LIN {X 0,Y 523.904,Z 128.222,A -85,B 0,C 180,E1 -4806.401,E2 -4806.401} C_VEL
LIN {X 0,Y 523.923,Z 128.218,A -85,B 0,C 180,E1 -4809.084,E2 -4809.084} C_VEL
LIN {X 0,Y 523.952,Z 128.218,A -85,B 0,C 180,E1 -4812.119,E2 -4812.119} C_VEL
LIN {X 0,Y 523.947,Z 128.218,A -85,B 0,C 180,E1 -4815.31,E2 -4815.31} C_VEL
LIN {X 0,Y 523.956,Z 128.214,A -85,B 0,C 180,E1 -4818.69,E2 -4818.69} C_VEL
LIN {X 0,Y 523.918,Z 128.221,A -85,B 0,C 180,E1 -4821.08,E2 -4821.08} C_VEL
LIN {X 0,Y 523.901,Z 128.225,A -85,B 0,C 180,E1 -4823.825,E2 -4823.825} C_VEL
LIN {X 0,Y 523.913,Z 128.219,A -85,B 0,C 180,E1 -4826.633,E2 -4826.633} C_VEL
LIN {X 0,Y 523.949,Z 128.223,A -85,B 0,C 180,E1 -4829.355,E2 -4829.355} C_VEL
LIN {X 0,Y 523.977,Z 128.211,A -85,B 0,C 180,E1 -4832.281,E2 -4832.281} C_VEL
LIN {X 0,Y 523.953,Z 128.215,A -85,B 0,C 180,E1 -4834.581,E2 -4834.581} C_VEL
LIN {X 0,Y 523.912,Z 128.227,A -85,B 0,C 180,E1 -4837.106,E2 -4837.106} C_VEL
LIN {X 0,Y 523.979,Z 128.211,A -85,B 0,C 180,E1 -4839.866,E2 -4839.866} C_VEL
LIN {X 0,Y 523.956,Z 128.219,A -85,B 0,C 180,E1 -4842.837,E2 -4842.837} C_VEL
LIN {X 0,Y 523.978,Z 128.217,A -85,B 0,C 180,E1 -4845.236,E2 -4845.236} C_VEL
LIN {X 0,Y 524.013,Z 128.208,A -85,B 0,C 180,E1 -4848.394,E2 -4848.394} C_VEL
LIN {X 0,Y 523.988,Z 128.211,A -85,B 0,C 180,E1 -4851.516,E2 -4851.516} C_VEL
LIN {X 0,Y 524.08,Z 128.204,A -85,B 0,C 180,E1 -4854.613,E2 -4854.613} C_VEL
LIN {X 0,Y 524.112,Z 128.194,A -85,B 0,C 180,E1 -4857.694,E2 -4857.694} C_VEL
LIN {X 0,Y 524.123,Z 128.2,A -85,B 0,C 180,E1 -4860.768,E2 -4860.768} C_VEL
LIN {X 0,Y 524.069,Z 128.202,A -85,B 0,C 180,E1 -4863.075,E2 -4863.075} C_VEL
LIN {X 0,Y 524.037,Z 128.207,A -85,B 0,C 180,E1 -4866.159,E2 -4866.159} C_VEL
LIN {X 0,Y 524,Z 128.217,A -85,B 0,C 180,E1 -4868.484,E2 -4868.484} C_VEL
LIN {X 0,Y 524.003,Z 128.209,A -85,B 0,C 180,E1 -4871.739,E2 -4871.739} C_VEL
LIN {X 0,Y 523.993,Z 128.21,A -85,B 0,C 180,E1 -4875.052,E2 -4875.052} C_VEL
LIN {X 0,Y 523.947,Z 128.219,A -85,B 0,C 180,E1 -4877.969,E2 -4877.969} C_VEL
LIN {X 0,Y 523.971,Z 128.218,A -85,B 0,C 180,E1 -4880.41,E2 -4880.41} C_VEL
LIN {X 0,Y 523.91,Z 128.22,A -85,B 0,C 180,E1 -4882.893,E2 -4882.893} C_VEL
LIN {X 0,Y 523.983,Z 128.218,A -85,B 0,C 180,E1 -4886.02,E2 -4886.02} C_VEL
LIN {X 0,Y 523.928,Z 128.217,A -85,B 0,C 180,E1 -4888.875,E2 -4888.875} C_VEL
LIN {X 0,Y 523.92,Z 128.221,A -85,B 0,C 180,E1 -4891.544,E2 -4891.544} C_VEL
LIN {X 0,Y 523.932,Z 128.22,A -85,B 0,C 180,E1 -4894.29,E2 -4894.29} C_VEL
LIN {X 0,Y 523.906,Z 128.221,A -85,B 0,C 180,E1 -4897.132,E2 -4897.132} C_VEL
LIN {X 0,Y 523.937,Z 128.22,A -85,B 0,C 180,E1 -4900.13,E2 -4900.13} C_VEL
LIN {X 0,Y 523.92,Z 128.22,A -85,B 0,C 180,E1 -4903.167,E2 -4903.167} C_VEL
LIN {X 0,Y 523.935,Z 128.223,A -85,B 0,C 180,E1 -4905.772,E2 -4905.772} C_VEL
LIN {X 0,Y 523.918,Z 128.219,A -85,B 0,C 180,E1 -4906.912,E2 -4906.912} C_VEL
LIN {X 0,Y 523.25,Z 128.31,A -85,B 0,C 180,E1 -4907.554,E2 -4907.554} C_VEL
LIN {X 0,Y 520.408,Z 128.661,A -85,B 0,C 180,E1 -4908.596,E2 -4908.596} C_VEL
LIN {X 0,Y 518.004,Z 128.962,A -85,B 0,C 180,E1 -4909.434,E2 -4909.434} C_VEL
LIN {X 0,Y 516.967,Z 129.086,A -85,B 0,C 180,E1 -4910.082,E2 -4910.082} C_VEL
LIN {X 0,Y 516.88,Z 129.096,A -85,B 0,C 180,E1 -4910.301,E2 -4910.301} C_VEL
LIN {X 0,Y 516.876,Z 129.103,A -85,B 0,C 180,E1 -4913.343,E2 -4913.343} C_VEL
LIN {X 0,Y 516.883,Z 129.095,A -85,B 0,C 180,E1 -4916.119,E2 -4916.119} C_VEL
LIN {X 0,Y 516.889,Z 129.097,A -85,B 0,C 180,E1 -4918.936,E2 -4918.936} C_VEL
LIN {X 0,Y 516.915,Z 129.095,A -85,B 0,C 180,E1 -4921.585,E2 -4921.585} C_VEL
LIN {X 0,Y 516.931,Z 129.089,A -85,B 0,C 180,E1 -4924.211,E2 -4924.211} C_VEL
LIN {X 0,Y 516.864,Z 129.101,A -85,B 0,C 180,E1 -4926.776,E2 -4926.776} C_VEL
LIN {X 0,Y 516.939,Z 129.089,A -85,B 0,C 180,E1 -4929.732,E2 -4929.732} C_VEL
LIN {X 0,Y 516.906,Z 129.095,A -85,B 0,C 180,E1 -4932.596,E2 -4932.596} C_VEL
LIN {X 0,Y 516.941,Z 129.096,A -85,B 0,C 180,E1 -4935.03,E2 -4935.03} C_VEL
LIN {X 0,Y 516.966,Z 129.085,A -85,B 0,C 180,E1 -4938.234,E2 -4938.234} C_VEL
LIN {X 0,Y 516.956,Z 129.087,A -85,B 0,C 180,E1 -4941.4,E2 -4941.4} C_VEL
LIN {X 0,Y 517.027,Z 129.082,A -85,B 0,C 180,E1 -4944.54,E2 -4944.54} C_VEL
LIN {X 0,Y 517.084,Z 129.072,A -85,B 0,C 180,E1 -4947.663,E2 -4947.663} C_VEL
LIN {X 0,Y 517.089,Z 129.079,A -85,B 0,C 180,E1 -4950.779,E2 -4950.779} C_VEL
LIN {X 0,Y 517.058,Z 129.277,A -85,B 0,C 180,E1 -4950.925,E2 -4950.925} C_VEL
LIN {X 0,Y 517.506,Z 134.385,A -85,B 0,C 180,E1 -4951.946,E2 -4951.946} C_VEL
LIN {X 0,Y 517.261,Z 148.661,A -85,B 0,C 180,E1 -4954.701,E2 -4954.701} C_VEL
LIN {X 0,Y 519.14,Z 158.814,A -85,B 0,C 180,E1 -4954.902,E2 -4954.902} C_VEL
LIN {X 0,Y 518.601,Z 255.581,A -85,B 0,C 180,E1 -4956.273,E2 -4956.273} C_VEL
LIN {X 0,Y 518.422,Z 269.344,A -85,B 0,C 180,E1 -4956.642,E2 -4956.642} C_VEL
LIN {X 0,Y 518.231,Z 280.872,A -85,B 0,C 180,E1 -4957.097,E2 -4957.097} C_VEL
LIN {X 0,Y 518.001,Z 292.37,A -85,B 0,C 180,E1 -4957.702,E2 -4957.702} C_VEL
LIN {X 0,Y 517.716,Z 303.803,A -85,B 0,C 180,E1 -4958.48,E2 -4958.48} C_VEL
LIN {X 0,Y 517.374,Z 314.408,A -85,B 0,C 180,E1 -4959.382,E2 -4959.382} C_VEL
LIN {X 0,Y 517.083,Z 323.83,A -85,B 0,C 180,E1 -4960.375,E2 -4960.375} C_VEL
LIN {X 0,Y 516.843,Z 333.07,A -85,B 0,C 180,E1 -4961.592,E2 -4961.592} C_VEL
LIN {X 0,Y 516.622,Z 340.269,A -85,B 0,C 180,E1 -4962.772,E2 -4962.772} C_VEL
LIN {X 0,Y 516.533,Z 345.22,A -85,B 0,C 180,E1 -4963.775,E2 -4963.775} C_VEL
LIN {X 0,Y 516.432,Z 350.035,A -85,B 0,C 180,E1 -4964.985,E2 -4964.985} C_VEL
LIN {X 0,Y 516.314,Z 353.712,A -85,B 0,C 180,E1 -4966.203,E2 -4966.203} C_VEL
LIN {X 0,Y 516.245,Z 356.678,A -85,B 0,C 180,E1 -4967.644,E2 -4967.644} C_VEL
LIN {X 0,Y 516.206,Z 358.228,A -85,B 0,C 180,E1 -4969.072,E2 -4969.072} C_VEL
LIN {X 0,Y 516.228,Z 358.561,A -85,B 0,C 180,E1 -4970.053,E2 -4970.053} C_VEL
LIN {X 0,Y 516.211,Z 357.794,A -85,B 0,C 180,E1 -4971.567,E2 -4971.567} C_VEL
LIN {X 0,Y 516.252,Z 356.747,A -85,B 0,C 180,E1 -4972.407,E2 -4972.407} C_VEL
LIN {X 0,Y 516.322,Z 354.262,A -85,B 0,C 180,E1 -4973.675,E2 -4973.675} C_VEL
LIN {X 0,Y 516.407,Z 350.603,A -85,B 0,C 180,E1 -4974.954,E2 -4974.954} C_VEL
LIN {X 0,Y 516.519,Z 345.117,A -85,B 0,C 180,E1 -4976.348,E2 -4976.348} C_VEL
LIN {X 0,Y 516.664,Z 339.024,A -85,B 0,C 180,E1 -4977.548,E2 -4977.548} C_VEL
LIN {X 0,Y 516.848,Z 332.152,A -85,B 0,C 180,E1 -4978.641,E2 -4978.641} C_VEL
LIN {X 0,Y 517.083,Z 324.555,A -85,B 0,C 180,E1 -4979.635,E2 -4979.635} C_VEL
LIN {X 0,Y 517.367,Z 315.378,A -85,B 0,C 180,E1 -4980.624,E2 -4980.624} C_VEL
LIN {X 0,Y 517.6,Z 304.961,A -85,B 0,C 180,E1 -4981.531,E2 -4981.531} C_VEL
LIN {X 0,Y 517.962,Z 293.968,A -85,B 0,C 180,E1 -4982.294,E2 -4982.294} C_VEL
LIN {X 0,Y 518.27,Z 281.601,A -85,B 0,C 180,E1 -4982.964,E2 -4982.964} C_VEL
LIN {X 0,Y 518.469,Z 268.694,A -85,B 0,C 180,E1 -4983.472,E2 -4983.472} C_VEL
LIN {X 0,Y 518.68,Z 255.806,A -85,B 0,C 180,E1 -4983.812,E2 -4983.812} C_VEL
LIN {X 0,Y 519.059,Z 157.607,A -85,B 0,C 180,E1 -4985.21,E2 -4985.21} C_VEL
LIN {X 0,Y 517.299,Z 148.488,A -85,B 0,C 180,E1 -4985.408,E2 -4985.408} C_VEL
LIN {X 0,Y 517.5,Z 133.51,A -85,B 0,C 180,E1 -4988.302,E2 -4988.302} C_VEL
LIN {X 0,Y 516.927,Z 129.098,A -85,B 0,C 180,E1 -4989.199,E2 -4989.199} C_VEL
LIN {X 0,Y 516.85,Z 129.105,A -85,B 0,C 180,E1 -4991.782,E2 -4991.782} C_VEL
LIN {X 0,Y 516.896,Z 129.102,A -85,B 0,C 180,E1 -4995.007,E2 -4995.007} C_VEL
LIN {X 0,Y 516.855,Z 129.102,A -85,B 0,C 180,E1 -4998.406,E2 -4998.406} C_VEL
LIN {X 0,Y 516.876,Z 129.103,A -85,B 0,C 180,E1 -5001.284,E2 -5001.284} C_VEL
LIN {X 0,Y 516.865,Z 129.096,A -85,B 0,C 180,E1 -5004.219,E2 -5004.219} C_VEL
LIN {X 0,Y 516.879,Z 129.104,A -85,B 0,C 180,E1 -5007.052,E2 -5007.052} C_VEL
LIN {X 0,Y 516.843,Z 129.102,A -85,B 0,C 180,E1 -5009.793,E2 -5009.793} C_VEL
LIN {X 0,Y 516.868,Z 129.103,A -85,B 0,C 180,E1 -5012.464,E2 -5012.464} C_VEL
LIN {X 0,Y 516.842,Z 129.105,A -85,B 0,C 180,E1 -5015.068,E2 -5015.068} C_VEL
LIN {X 0,Y 516.87,Z 129.095,A -85,B 0,C 180,E1 -5017.622,E2 -5017.622} C_VEL
LIN {X 0,Y 516.862,Z 129.102,A -85,B 0,C 180,E1 -5020.127,E2 -5020.127} C_VEL
LIN {X 0,Y 516.869,Z 129.104,A -85,B 0,C 180,E1 -5022.594,E2 -5022.594} C_VEL
LIN {X 0,Y 516.873,Z 129.096,A -85,B 0,C 180,E1 -5025.028,E2 -5025.028} C_VEL
LIN {X 0,Y 516.921,Z 129.096,A -85,B 0,C 180,E1 -5028.233,E2 -5028.233} C_VEL
LIN {X 0,Y 516.917,Z 129.092,A -85,B 0,C 180,E1 -5031.399,E2 -5031.399} C_VEL
LIN {X 0,Y 516.978,Z 129.085,A -85,B 0,C 180,E1 -5034.54,E2 -5034.54} C_VEL
LIN {X 0,Y 517.073,Z 129.075,A -85,B 0,C 180,E1 -5037.663,E2 -5037.663} C_VEL
LIN {X 0,Y 517.066,Z 129.079,A -85,B 0,C 180,E1 -5040,E2 -5040} C_VEL
LIN {X 0,Y 517.073,Z 129.07,A -85,B 0,C 180,E1 -5042.337,E2 -5042.337} C_VEL
LIN {X 0,Y 516.969,Z 129.085,A -85,B 0,C 180,E1 -5046.244,E2 -5046.244} C_VEL
LIN {X 0,Y 516.913,Z 129.095,A -85,B 0,C 180,E1 -5049.39,E2 -5049.39} C_VEL
LIN {X 0,Y 516.955,Z 129.088,A -85,B 0,C 180,E1 -5051.807,E2 -5051.807} C_VEL
LIN {X 0,Y 516.939,Z 129.093,A -85,B 0,C 180,E1 -5055.143,E2 -5055.143} C_VEL
LIN {X 0,Y 516.88,Z 129.093,A -85,B 0,C 180,E1 -5058.224,E2 -5058.224} C_VEL
LIN {X 0,Y 516.907,Z 129.094,A -85,B 0,C 180,E1 -5060.702,E2 -5060.702} C_VEL
LIN {X 0,Y 516.887,Z 129.095,A -85,B 0,C 180,E1 -5064.073,E2 -5064.073} C_VEL
LIN {X 0,Y 516.896,Z 129.095,A -85,B 0,C 180,E1 -5066.66,E2 -5066.66} C_VEL
LIN {X 0,Y 516.888,Z 129.095,A -85,B 0,C 180,E1 -5069.519,E2 -5069.519} C_VEL
LIN {X 0,Y 516.896,Z 129.098,A -85,B 0,C 180,E1 -5072.543,E2 -5072.543} C_VEL
LIN {X 0,Y 516.867,Z 129.1,A -85,B 0,C 180,E1 -5075.329,E2 -5075.329} C_VEL
LIN {X 0,Y 516.881,Z 129.095,A -85,B 0,C 180,E1 -5077.943,E2 -5077.943} C_VEL
LIN {X 0,Y 516.866,Z 129.105,A -85,B 0,C 180,E1 -5080.744,E2 -5080.744} C_VEL
LIN {X 0,Y 516.857,Z 129.104,A -85,B 0,C 180,E1 -5082.834,E2 -5082.834} C_VEL
LIN {X 0,Y 516.898,Z 129.096,A -85,B 0,C 180,E1 -5085.007,E2 -5085.007} C_VEL
LIN {X 0,Y 516.911,Z 129.101,A -85,B 0,C 180,E1 -5088.4,E2 -5088.4} C_VEL
LIN {X 0,Y 516.883,Z 129.096,A -85,B 0,C 180,E1 -5091.284,E2 -5091.284} C_VEL
LIN {X 0,Y 516.87,Z 129.105,A -85,B 0,C 180,E1 -5094.219,E2 -5094.219} C_VEL
LIN {X 0,Y 516.898,Z 129.095,A -85,B 0,C 180,E1 -5097.053,E2 -5097.053} C_VEL
LIN {X 0,Y 516.889,Z 129.101,A -85,B 0,C 180,E1 -5099.796,E2 -5099.796} C_VEL
LIN {X 0,Y 516.925,Z 129.095,A -85,B 0,C 180,E1 -5102.467,E2 -5102.467} C_VEL
LIN {X 0,Y 516.941,Z 129.15,A -85,B 0,C 180,E1 -5104.939,E2 -5104.939} C_VEL
LIN {X 0,Y 518.489,Z 138.225,A -85,B 0,C 180,E1 -5106.43,E2 -5106.43} C_VEL
LIN {X 0,Y 517.938,Z 158.539,A -85,B 0,C 180,E1 -5109.543,E2 -5109.543} C_VEL
LIN {X 0,Y 517.506,Z 178.873,A -85,B 0,C 180,E1 -5112.616,E2 -5112.616} C_VEL
LIN {X 0,Y 517.216,Z 192.296,A -85,B 0,C 180,E1 -5114.623,E2 -5114.623} C_VEL
LIN {X 0,Y 519.028,Z 206.259,A -85,B 0,C 180,E1 -5114.878,E2 -5114.878} C_VEL
LIN {X 0,Y 518.589,Z 300.529,A -85,B 0,C 180,E1 -5116.206,E2 -5116.206} C_VEL
LIN {X 0,Y 518.322,Z 313.972,A -85,B 0,C 180,E1 -5116.548,E2 -5116.548} C_VEL
LIN {X 0,Y 518.034,Z 327.363,A -85,B 0,C 180,E1 -5117.065,E2 -5117.065} C_VEL
LIN {X 0,Y 517.778,Z 338.798,A -85,B 0,C 180,E1 -5117.668,E2 -5117.668} C_VEL
LIN {X 0,Y 517.447,Z 350.26,A -85,B 0,C 180,E1 -5118.443,E2 -5118.443} C_VEL
LIN {X 0,Y 517.191,Z 360.762,A -85,B 0,C 180,E1 -5119.33,E2 -5119.33} C_VEL
LIN {X 0,Y 516.899,Z 369.348,A -85,B 0,C 180,E1 -5120.215,E2 -5120.215} C_VEL
LIN {X 0,Y 516.68,Z 377.273,A -85,B 0,C 180,E1 -5121.198,E2 -5121.198} C_VEL
LIN {X 0,Y 516.516,Z 385.017,A -85,B 0,C 180,E1 -5122.376,E2 -5122.376} C_VEL
LIN {X 0,Y 516.374,Z 392.154,A -85,B 0,C 180,E1 -5123.749,E2 -5123.749} C_VEL
LIN {X 0,Y 516.312,Z 396.906,A -85,B 0,C 180,E1 -5124.924,E2 -5124.924} C_VEL
LIN {X 0,Y 516.352,Z 400.54,A -85,B 0,C 180,E1 -5126.098,E2 -5126.098} C_VEL
LIN {X 0,Y 516.303,Z 402.413,A -85,B 0,C 180,E1 -5126.879,E2 -5126.879} C_VEL
LIN {X 0,Y 516.264,Z 403.816,A -85,B 0,C 180,E1 -5127.659,E2 -5127.659} C_VEL
LIN {X 0,Y 516.172,Z 405.43,A -85,B 0,C 180,E1 -5129.22,E2 -5129.22} C_VEL
LIN {X 0,Y 516.173,Z 405.651,A -85,B 0,C 180,E1 -5130,E2 -5130} C_VEL
LIN {X 0,Y 516.193,Z 404.829,A -85,B 0,C 180,E1 -5131.56,E2 -5131.56} C_VEL
LIN {X 0,Y 516.264,Z 403.835,A -85,B 0,C 180,E1 -5132.34,E2 -5132.34} C_VEL
LIN {X 0,Y 516.303,Z 402.436,A -85,B 0,C 180,E1 -5133.121,E2 -5133.121} C_VEL
LIN {X 0,Y 516.31,Z 399.49,A -85,B 0,C 180,E1 -5134.293,E2 -5134.293} C_VEL
LIN {X 0,Y 516.367,Z 395.502,A -85,B 0,C 180,E1 -5135.467,E2 -5135.467} C_VEL
LIN {X 0,Y 516.427,Z 389.355,A -85,B 0,C 180,E1 -5136.84,E2 -5136.84} C_VEL
LIN {X 0,Y 516.567,Z 382.66,A -85,B 0,C 180,E1 -5138.016,E2 -5138.016} C_VEL
LIN {X 0,Y 516.755,Z 374.344,A -85,B 0,C 180,E1 -5139.195,E2 -5139.195} C_VEL
LIN {X 0,Y 516.985,Z 365.818,A -85,B 0,C 180,E1 -5140.179,E2 -5140.179} C_VEL
LIN {X 0,Y 517.301,Z 355.287,A -85,B 0,C 180,E1 -5141.163,E2 -5141.163} C_VEL
LIN {X 0,Y 517.621,Z 343.415,A -85,B 0,C 180,E1 -5142.051,E2 -5142.051} C_VEL
LIN {X 0,Y 517.947,Z 331.506,A -85,B 0,C 180,E1 -5142.738,E2 -5142.738} C_VEL
LIN {X 0,Y 518.211,Z 319.097,A -85,B 0,C 180,E1 -5143.28,E2 -5143.28} C_VEL
LIN {X 0,Y 518.484,Z 306.333,A -85,B 0,C 180,E1 -5143.672,E2 -5143.672} C_VEL
LIN {X 0,Y 518.634,Z 291.09,A -85,B 0,C 180,E1 -5143.943,E2 -5143.943} C_VEL
LIN {X 0,Y 518.97,Z 204.341,A -85,B 0,C 180,E1 -5145.152,E2 -5145.152} C_VEL
LIN {X 0,Y 517.23,Z 192.384,A -85,B 0,C 180,E1 -5145.39,E2 -5145.39} C_VEL
LIN {X 0,Y 517.621,Z 174.235,A -85,B 0,C 180,E1 -5148.116,E2 -5148.116} C_VEL
LIN {X 0,Y 518.165,Z 152.086,A -85,B 0,C 180,E1 -5151.482,E2 -5151.482} C_VEL
LIN {X 0,Y 518.451,Z 137.182,A -85,B 0,C 180,E1 -5153.783,E2 -5153.783} C_VEL
LIN {X 0,Y 516.924,Z 129.096,A -85,B 0,C 180,E1 -5155.142,E2 -5155.142} C_VEL
LIN {X 0,Y 516.918,Z 129.099,A -85,B 0,C 180,E1 -5157.903,E2 -5157.903} C_VEL
LIN {X 0,Y 516.894,Z 129.102,A -85,B 0,C 180,E1 -5160.203,E2 -5160.203} C_VEL
LIN {X 0,Y 516.896,Z 129.093,A -85,B 0,C 180,E1 -5162.947,E2 -5162.947} C_VEL
LIN {X 0,Y 516.872,Z 129.103,A -85,B 0,C 180,E1 -5165.78,E2 -5165.78} C_VEL
LIN {X 0,Y 516.883,Z 129.095,A -85,B 0,C 180,E1 -5168.716,E2 -5168.716} C_VEL
LIN {X 0,Y 516.913,Z 129.1,A -85,B 0,C 180,E1 -5171.775,E2 -5171.775} C_VEL
LIN {X 0,Y 516.896,Z 129.094,A -85,B 0,C 180,E1 -5175.007,E2 -5175.007} C_VEL
LIN {X 0,Y 516.914,Z 129.091,A -85,B 0,C 180,E1 -5178.399,E2 -5178.399} C_VEL
LIN {X 0,Y 516.881,Z 129.1,A -85,B 0,C 180,E1 -5181.284,E2 -5181.284} C_VEL
LIN {X 0,Y 516.871,Z 129.097,A -85,B 0,C 180,E1 -5184.219,E2 -5184.219} C_VEL
LIN {X 0,Y 516.881,Z 129.098,A -85,B 0,C 180,E1 -5187.052,E2 -5187.052} C_VEL
LIN {X 0,Y 516.887,Z 129.097,A -85,B 0,C 180,E1 -5189.796,E2 -5189.796} C_VEL
LIN {X 0,Y 516.926,Z 129.09,A -85,B 0,C 180,E1 -5192.467,E2 -5192.467} C_VEL
LIN {X 0,Y 516.909,Z 129.098,A -85,B 0,C 180,E1 -5195.072,E2 -5195.072} C_VEL
LIN {X 0,Y 516.886,Z 129.095,A -85,B 0,C 180,E1 -5198.462,E2 -5198.462} C_VEL
LIN {X 0,Y 516.9,Z 129.099,A -85,B 0,C 180,E1 -5200.955,E2 -5200.955} C_VEL
LIN {X 0,Y 516.907,Z 129.096,A -85,B 0,C 180,E1 -5203.41,E2 -5203.41} C_VEL
LIN {X 0,Y 516.894,Z 129.094,A -85,B 0,C 180,E1 -5205.833,E2 -5205.833} C_VEL
LIN {X 0,Y 516.966,Z 129.085,A -85,B 0,C 180,E1 -5208.234,E2 -5208.234} C_VEL
LIN {X 0,Y 516.956,Z 129.088,A -85,B 0,C 180,E1 -5211.399,E2 -5211.399} C_VEL
LIN {X 0,Y 517.027,Z 129.082,A -85,B 0,C 180,E1 -5214.54,E2 -5214.54} C_VEL
LIN {X 0,Y 517.084,Z 129.07,A -85,B 0,C 180,E1 -5217.663,E2 -5217.663} C_VEL
LIN {X 0,Y 517.093,Z 129.076,A -85,B 0,C 180,E1 -5220.779,E2 -5220.779} C_VEL
LIN {X 0,Y 517.01,Z 129.081,A -85,B 0,C 180,E1 -5223.117,E2 -5223.117} C_VEL
LIN {X 0,Y 517.002,Z 129.084,A -85,B 0,C 180,E1 -5226.243,E2 -5226.243} C_VEL
LIN {X 0,Y 516.945,Z 129.087,A -85,B 0,C 180,E1 -5229.389,E2 -5229.389} C_VEL
LIN {X 0,Y 516.952,Z 129.088,A -85,B 0,C 180,E1 -5231.807,E2 -5231.807} C_VEL
LIN {X 0,Y 516.944,Z 129.087,A -85,B 0,C 180,E1 -5235.146,E2 -5235.146} C_VEL
LIN {X 0,Y 516.915,Z 129.099,A -85,B 0,C 180,E1 -5238.222,E2 -5238.222} C_VEL
LIN {X 0,Y 516.912,Z 129.094,A -85,B 0,C 180,E1 -5240.701,E2 -5240.701} C_VEL
LIN {X 0,Y 516.89,Z 129.102,A -85,B 0,C 180,E1 -5244.073,E2 -5244.073} C_VEL
LIN {X 0,Y 516.921,Z 129.092,A -85,B 0,C 180,E1 -5246.658,E2 -5246.658} C_VEL
LIN {X 0,Y 516.909,Z 129.094,A -85,B 0,C 180,E1 -5249.523,E2 -5249.523} C_VEL
LIN {X 0,Y 516.895,Z 129.095,A -85,B 0,C 180,E1 -5252.543,E2 -5252.543} C_VEL
LIN {X 0,Y 516.865,Z 129.099,A -85,B 0,C 180,E1 -5255.33,E2 -5255.33} C_VEL
LIN {X 0,Y 516.88,Z 129.102,A -85,B 0,C 180,E1 -5257.943,E2 -5257.943} C_VEL
LIN {X 0,Y 516.882,Z 129.095,A -85,B 0,C 180,E1 -5260.742,E2 -5260.742} C_VEL
LIN {X 0,Y 516.883,Z 129.095,A -85,B 0,C 180,E1 -5262.831,E2 -5262.831} C_VEL
LIN {X 0,Y 516.882,Z 129.098,A -85,B 0,C 180,E1 -5266.097,E2 -5266.097} C_VEL
LIN {X 0,Y 516.912,Z 129.091,A -85,B 0,C 180,E1 -5268.399,E2 -5268.399} C_VEL
LIN {X 0,Y 516.88,Z 129.096,A -85,B 0,C 180,E1 -5270.301,E2 -5270.301} C_VEL
LIN {X 0,Y 516.209,Z 129.181,A -85,B 0,C 180,E1 -5270.952,E2 -5270.952} C_VEL
LIN {X 0,Y 513.362,Z 129.541,A -85,B 0,C 180,E1 -5272.007,E2 -5272.007} C_VEL
LIN {X 0,Y 510.952,Z 129.844,A -85,B 0,C 180,E1 -5272.857,E2 -5272.857} C_VEL
LIN {X 0,Y 509.909,Z 129.972,A -85,B 0,C 180,E1 -5273.514,E2 -5273.514} C_VEL
LIN {X 0,Y 509.819,Z 129.98,A -85,B 0,C 180,E1 -5273.736,E2 -5273.736} C_VEL
LIN {X 0,Y 509.841,Z 129.972,A -85,B 0,C 180,E1 -5276.538,E2 -5276.538} C_VEL
LIN {X 0,Y 509.842,Z 129.981,A -85,B 0,C 180,E1 -5279.334,E2 -5279.334} C_VEL
LIN {X 0,Y 509.889,Z 129.966,A -85,B 0,C 180,E1 -5282.054,E2 -5282.054} C_VEL
LIN {X 0,Y 509.875,Z 129.97,A -85,B 0,C 180,E1 -5284.704,E2 -5284.704} C_VEL
LIN {X 0,Y 509.826,Z 129.978,A -85,B 0,C 180,E1 -5287.458,E2 -5287.458} C_VEL
LIN {X 0,Y 509.916,Z 129.963,A -85,B 0,C 180,E1 -5289.845,E2 -5289.845} C_VEL
LIN {X 0,Y 509.873,Z 129.975,A -85,B 0,C 180,E1 -5293.174,E2 -5293.174} C_VEL
LIN {X 0,Y 509.861,Z 129.971,A -85,B 0,C 180,E1 -5295.634,E2 -5295.634} C_VEL
LIN {X 0,Y 509.913,Z 129.972,A -85,B 0,C 180,E1 -5298.875,E2 -5298.875} C_VEL
LIN {X 0,Y 509.921,Z 129.963,A -85,B 0,C 180,E1 -5302.078,E2 -5302.078} C_VEL
LIN {X 0,Y 509.978,Z 129.959,A -85,B 0,C 180,E1 -5304.464,E2 -5304.464} C_VEL
LIN {X 0,Y 510.055,Z 129.948,A -85,B 0,C 180,E1 -5307.631,E2 -5307.631} C_VEL
LIN {X 0,Y 510.063,Z 129.964,A -85,B 0,C 180,E1 -5310.765,E2 -5310.765} C_VEL
LIN {X 0,Y 510.477,Z 136.956,A -85,B 0,C 180,E1 -5312.17,E2 -5312.17} C_VEL
LIN {X 0,Y 510.218,Z 148.664,A -85,B 0,C 180,E1 -5314.469,E2 -5314.469} C_VEL
LIN {X 0,Y 512.252,Z 159.199,A -85,B 0,C 180,E1 -5314.697,E2 -5314.697} C_VEL
LIN {X 0,Y 511.715,Z 255.843,A -85,B 0,C 180,E1 -5316.086,E2 -5316.086} C_VEL
LIN {X 0,Y 511.542,Z 269.612,A -85,B 0,C 180,E1 -5316.459,E2 -5316.459} C_VEL
LIN {X 0,Y 511.319,Z 281.983,A -85,B 0,C 180,E1 -5316.957,E2 -5316.957} C_VEL
LIN {X 0,Y 511.036,Z 294.579,A -85,B 0,C 180,E1 -5317.654,E2 -5317.654} C_VEL
LIN {X 0,Y 510.681,Z 306.516,A -85,B 0,C 180,E1 -5318.508,E2 -5318.508} C_VEL
LIN {X 0,Y 510.373,Z 315.527,A -85,B 0,C 180,E1 -5319.312,E2 -5319.312} C_VEL
LIN {X 0,Y 510.056,Z 324.771,A -85,B 0,C 180,E1 -5320.319,E2 -5320.319} C_VEL
LIN {X 0,Y 509.819,Z 333.265,A -85,B 0,C 180,E1 -5321.458,E2 -5321.458} C_VEL
LIN {X 0,Y 509.572,Z 341.006,A -85,B 0,C 180,E1 -5322.749,E2 -5322.749} C_VEL
LIN {X 0,Y 509.439,Z 346.763,A -85,B 0,C 180,E1 -5323.971,E2 -5323.971} C_VEL
LIN {X 0,Y 509.331,Z 351.294,A -85,B 0,C 180,E1 -5325.199,E2 -5325.199} C_VEL
LIN {X 0,Y 509.257,Z 353.69,A -85,B 0,C 180,E1 -5326.022,E2 -5326.022} C_VEL
LIN {X 0,Y 509.187,Z 355.643,A -85,B 0,C 180,E1 -5326.849,E2 -5326.849} C_VEL
LIN {X 0,Y 509.151,Z 357.186,A -85,B 0,C 180,E1 -5327.743,E2 -5327.743} C_VEL
LIN {X 0,Y 509.137,Z 358.725,A -85,B 0,C 180,E1 -5329.347,E2 -5329.347} C_VEL
LIN {X 0,Y 509.139,Z 358.863,A -85,B 0,C 180,E1 -5330.188,E2 -5330.188} C_VEL
LIN {X 0,Y 509.116,Z 358.558,A -85,B 0,C 180,E1 -5331.034,E2 -5331.034} C_VEL
LIN {X 0,Y 509.162,Z 357.182,A -85,B 0,C 180,E1 -5332.361,E2 -5332.361} C_VEL
LIN {X 0,Y 509.282,Z 353.923,A -85,B 0,C 180,E1 -5333.991,E2 -5333.991} C_VEL
LIN {X 0,Y 509.36,Z 349.87,A -85,B 0,C 180,E1 -5335.324,E2 -5335.324} C_VEL
LIN {X 0,Y 509.498,Z 344.542,A -85,B 0,C 180,E1 -5336.635,E2 -5336.635} C_VEL
LIN {X 0,Y 509.697,Z 337.609,A -85,B 0,C 180,E1 -5337.957,E2 -5337.957} C_VEL
LIN {X 0,Y 509.919,Z 330.307,A -85,B 0,C 180,E1 -5339.067,E2 -5339.067} C_VEL
LIN {X 0,Y 510.217,Z 320.57,A -85,B 0,C 180,E1 -5340.264,E2 -5340.264} C_VEL
LIN {X 0,Y 510.521,Z 311.039,A -85,B 0,C 180,E1 -5341.207,E2 -5341.207} C_VEL
LIN {X 0,Y 510.863,Z 299.789,A -85,B 0,C 180,E1 -5342.098,E2 -5342.098} C_VEL
LIN {X 0,Y 511.253,Z 288.591,A -85,B 0,C 180,E1 -5342.799,E2 -5342.799} C_VEL
LIN {X 0,Y 511.454,Z 277.444,A -85,B 0,C 180,E1 -5343.343,E2 -5343.343} C_VEL
LIN {X 0,Y 511.674,Z 264.471,A -85,B 0,C 180,E1 -5343.799,E2 -5343.799} C_VEL
LIN {X 0,Y 511.825,Z 250.828,A -85,B 0,C 180,E1 -5344.099,E2 -5344.099} C_VEL
LIN {X 0,Y 512.207,Z 158.542,A -85,B 0,C 180,E1 -5345.414,E2 -5345.414} C_VEL
LIN {X 0,Y 510.334,Z 148.724,A -85,B 0,C 180,E1 -5345.637,E2 -5345.637} C_VEL
LIN {X 0,Y 510.515,Z 135.005,A -85,B 0,C 180,E1 -5348.308,E2 -5348.308} C_VEL
LIN {X 0,Y 509.87,Z 129.977,A -85,B 0,C 180,E1 -5349.35,E2 -5349.35} C_VEL
LIN {X 0,Y 509.791,Z 129.981,A -85,B 0,C 180,E1 -5352.494,E2 -5352.494} C_VEL
LIN {X 0,Y 509.839,Z 129.981,A -85,B 0,C 180,E1 -5355.33,E2 -5355.33} C_VEL
LIN {X 0,Y 509.807,Z 129.981,A -85,B 0,C 180,E1 -5358.57,E2 -5358.57} C_VEL
LIN {X 0,Y 509.849,Z 129.974,A -85,B 0,C 180,E1 -5361.787,E2 -5361.787} C_VEL
LIN {X 0,Y 509.824,Z 129.977,A -85,B 0,C 180,E1 -5364.622,E2 -5364.622} C_VEL
LIN {X 0,Y 509.857,Z 129.973,A -85,B 0,C 180,E1 -5367.481,E2 -5367.481} C_VEL
LIN {X 0,Y 509.827,Z 129.978,A -85,B 0,C 180,E1 -5370.28,E2 -5370.28} C_VEL
LIN {X 0,Y 509.816,Z 129.982,A -85,B 0,C 180,E1 -5372.941,E2 -5372.941} C_VEL
LIN {X 0,Y 509.823,Z 129.976,A -85,B 0,C 180,E1 -5375.572,E2 -5375.572} C_VEL
LIN {X 0,Y 509.799,Z 129.979,A -85,B 0,C 180,E1 -5378.148,E2 -5378.148} C_VEL
LIN {X 0,Y 509.806,Z 129.981,A -85,B 0,C 180,E1 -5380.679,E2 -5380.679} C_VEL
LIN {X 0,Y 509.786,Z 129.98,A -85,B 0,C 180,E1 -5383.172,E2 -5383.172} C_VEL
LIN {X 0,Y 509.813,Z 129.975,A -85,B 0,C 180,E1 -5385.633,E2 -5385.633} C_VEL
LIN {X 0,Y 509.889,Z 129.974,A -85,B 0,C 180,E1 -5388.132,E2 -5388.132} C_VEL
LIN {X 0,Y 509.871,Z 129.969,A -85,B 0,C 180,E1 -5391.279,E2 -5391.279} C_VEL
LIN {X 0,Y 509.915,Z 129.964,A -85,B 0,C 180,E1 -5393.67,E2 -5393.67} C_VEL
LIN {X 0,Y 509.882,Z 129.966,A -85,B 0,C 180,E1 -5396.84,E2 -5396.84} C_VEL
LIN {X 0,Y 509.922,Z 129.962,A -85,B 0,C 180,E1 -5398.421,E2 -5398.421} C_VEL
LIN {X 0,Y 510.035,Z 129.955,A -85,B 0,C 180,E1 -5400,E2 -5400} C_VEL
LIN {X 0,Y 510.042,Z 129.945,A -85,B 0,C 180,E1 -5402.369,E2 -5402.369} C_VEL
LIN {X 0,Y 509.937,Z 129.966,A -85,B 0,C 180,E1 -5405.536,E2 -5405.536} C_VEL
LIN {X 0,Y 509.879,Z 129.97,A -85,B 0,C 180,E1 -5407.923,E2 -5407.923} C_VEL
LIN {X 0,Y 509.913,Z 129.967,A -85,B 0,C 180,E1 -5411.126,E2 -5411.126} C_VEL
LIN {X 0,Y 509.847,Z 129.971,A -85,B 0,C 180,E1 -5414.367,E2 -5414.367} C_VEL
LIN {X 0,Y 509.847,Z 129.973,A -85,B 0,C 180,E1 -5416.827,E2 -5416.827} C_VEL
LIN {X 0,Y 509.917,Z 129.963,A -85,B 0,C 180,E1 -5420.155,E2 -5420.155} C_VEL
LIN {X 0,Y 509.82,Z 129.978,A -85,B 0,C 180,E1 -5423.564,E2 -5423.564} C_VEL
LIN {X 0,Y 509.877,Z 129.967,A -85,B 0,C 180,E1 -5426.37,E2 -5426.37} C_VEL
LIN {X 0,Y 509.854,Z 129.97,A -85,B 0,C 180,E1 -5429.752,E2 -5429.752} C_VEL
LIN {X 0,Y 509.869,Z 129.977,A -85,B 0,C 180,E1 -5432.773,E2 -5432.773} C_VEL
LIN {X 0,Y 509.827,Z 129.975,A -85,B 0,C 180,E1 -5435.578,E2 -5435.578} C_VEL
LIN {X 0,Y 509.85,Z 129.974,A -85,B 0,C 180,E1 -5438.338,E2 -5438.338} C_VEL
LIN {X 0,Y 509.846,Z 129.973,A -85,B 0,C 180,E1 -5441.427,E2 -5441.427} C_VEL
LIN {X 0,Y 509.841,Z 129.98,A -85,B 0,C 180,E1 -5444.67,E2 -5444.67} C_VEL
LIN {X 0,Y 509.851,Z 129.978,A -85,B 0,C 180,E1 -5448.104,E2 -5448.104} C_VEL
LIN {X 0,Y 509.849,Z 129.977,A -85,B 0,C 180,E1 -5450.648,E2 -5450.648} C_VEL
LIN {X 0,Y 509.812,Z 129.978,A -85,B 0,C 180,E1 -5453.646,E2 -5453.646} C_VEL
LIN {X 0,Y 509.862,Z 129.975,A -85,B 0,C 180,E1 -5456.539,E2 -5456.539} C_VEL
LIN {X 0,Y 509.845,Z 129.976,A -85,B 0,C 180,E1 -5459.334,E2 -5459.334} C_VEL
LIN {X 0,Y 509.886,Z 129.975,A -85,B 0,C 180,E1 -5462.054,E2 -5462.054} C_VEL
LIN {X 0,Y 509.895,Z 130.039,A -85,B 0,C 180,E1 -5464.753,E2 -5464.753} C_VEL
LIN {X 0,Y 511.556,Z 139.292,A -85,B 0,C 180,E1 -5466.306,E2 -5466.306} C_VEL
LIN {X 0,Y 510.995,Z 159.023,A -85,B 0,C 180,E1 -5469.376,E2 -5469.376} C_VEL
LIN {X 0,Y 510.5,Z 179.915,A -85,B 0,C 180,E1 -5472.576,E2 -5472.576} C_VEL
LIN {X 0,Y 510.239,Z 192.104,A -85,B 0,C 180,E1 -5474.409,E2 -5474.409} C_VEL
LIN {X 0,Y 512.181,Z 206.837,A -85,B 0,C 180,E1 -5474.681,E2 -5474.681} C_VEL
LIN {X 0,Y 511.709,Z 300.168,A -85,B 0,C 180,E1 -5476.017,E2 -5476.017} C_VEL
LIN {X 0,Y 511.463,Z 312.843,A -85,B 0,C 180,E1 -5476.339,E2 -5476.339} C_VEL
LIN {X 0,Y 511.123,Z 325.863,A -85,B 0,C 180,E1 -5476.836,E2 -5476.836} C_VEL
LIN {X 0,Y 510.821,Z 337.563,A -85,B 0,C 180,E1 -5477.443,E2 -5477.443} C_VEL
LIN {X 0,Y 510.509,Z 348.608,A -85,B 0,C 180,E1 -5478.183,E2 -5478.183} C_VEL
LIN {X 0,Y 510.187,Z 359.336,A -85,B 0,C 180,E1 -5479.081,E2 -5479.081} C_VEL
LIN {X 0,Y 509.843,Z 369.002,A -85,B 0,C 180,E1 -5480.078,E2 -5480.078} C_VEL
LIN {X 0,Y 509.64,Z 376.932,A -85,B 0,C 180,E1 -5481.075,E2 -5481.075} C_VEL
LIN {X 0,Y 509.429,Z 384.679,A -85,B 0,C 180,E1 -5482.27,E2 -5482.27} C_VEL
LIN {X 0,Y 509.309,Z 390.998,A -85,B 0,C 180,E1 -5483.483,E2 -5483.483} C_VEL
LIN {X 0,Y 509.241,Z 396.575,A -85,B 0,C 180,E1 -5484.853,E2 -5484.853} C_VEL
LIN {X 0,Y 509.246,Z 400.211,A -85,B 0,C 180,E1 -5486.043,E2 -5486.043} C_VEL
LIN {X 0,Y 509.219,Z 402.086,A -85,B 0,C 180,E1 -5486.835,E2 -5486.835} C_VEL
LIN {X 0,Y 509.193,Z 403.491,A -85,B 0,C 180,E1 -5487.627,E2 -5487.627} C_VEL
LIN {X 0,Y 509.085,Z 405.106,A -85,B 0,C 180,E1 -5489.209,E2 -5489.209} C_VEL
LIN {X 0,Y 509.083,Z 405.327,A -85,B 0,C 180,E1 -5490,E2 -5490} C_VEL
LIN {X 0,Y 509.113,Z 404.507,A -85,B 0,C 180,E1 -5491.582,E2 -5491.582} C_VEL
LIN {X 0,Y 509.193,Z 403.513,A -85,B 0,C 180,E1 -5492.373,E2 -5492.373} C_VEL
LIN {X 0,Y 509.219,Z 402.113,A -85,B 0,C 180,E1 -5493.165,E2 -5493.165} C_VEL
LIN {X 0,Y 509.203,Z 399.166,A -85,B 0,C 180,E1 -5494.353,E2 -5494.353} C_VEL
LIN {X 0,Y 509.277,Z 395.177,A -85,B 0,C 180,E1 -5495.543,E2 -5495.543} C_VEL
LIN {X 0,Y 509.343,Z 389.14,A -85,B 0,C 180,E1 -5496.914,E2 -5496.914} C_VEL
LIN {X 0,Y 509.493,Z 382.333,A -85,B 0,C 180,E1 -5498.128,E2 -5498.128} C_VEL
LIN {X 0,Y 509.716,Z 374.015,A -85,B 0,C 180,E1 -5499.323,E2 -5499.323} C_VEL
LIN {X 0,Y 509.957,Z 365.486,A -85,B 0,C 180,E1 -5500.321,E2 -5500.321} C_VEL
LIN {X 0,Y 510.299,Z 354.952,A -85,B 0,C 180,E1 -5501.318,E2 -5501.318} C_VEL
LIN {X 0,Y 510.617,Z 343.942,A -85,B 0,C 180,E1 -5502.158,E2 -5502.158} C_VEL
LIN {X 0,Y 510.979,Z 333.109,A -85,B 0,C 180,E1 -5502.814,E2 -5502.814} C_VEL
LIN {X 0,Y 511.243,Z 321.351,A -85,B 0,C 180,E1 -5503.363,E2 -5503.363} C_VEL
LIN {X 0,Y 511.542,Z 307.809,A -85,B 0,C 180,E1 -5503.81,E2 -5503.81} C_VEL
LIN {X 0,Y 511.764,Z 294.248,A -85,B 0,C 180,E1 -5504.083,E2 -5504.083} C_VEL
LIN {X 0,Y 511.999,Z 204.487,A -85,B 0,C 180,E1 -5505.357,E2 -5505.357} C_VEL
LIN {X 0,Y 510.203,Z 192.079,A -85,B 0,C 180,E1 -5505.604,E2 -5505.604} C_VEL
LIN {X 0,Y 510.736,Z 172.018,A -85,B 0,C 180,E1 -5508.659,E2 -5508.659} C_VEL
LIN {X 0,Y 511.282,Z 150.396,A -85,B 0,C 180,E1 -5511.998,E2 -5511.998} C_VEL
LIN {X 0,Y 511.481,Z 138.206,A -85,B 0,C 180,E1 -5513.913,E2 -5513.913} C_VEL
LIN {X 0,Y 509.89,Z 129.973,A -85,B 0,C 180,E1 -5515.295,E2 -5515.295} C_VEL
LIN {X 0,Y 509.89,Z 129.975,A -85,B 0,C 180,E1 -5518.099,E2 -5518.099} C_VEL
LIN {X 0,Y 509.847,Z 129.974,A -85,B 0,C 180,E1 -5521.28,E2 -5521.28} C_VEL
LIN {X 0,Y 509.858,Z 129.975,A -85,B 0,C 180,E1 -5524.202,E2 -5524.202} C_VEL
LIN {X 0,Y 509.818,Z 129.977,A -85,B 0,C 180,E1 -5527.341,E2 -5527.341} C_VEL
LIN {X 0,Y 509.839,Z 129.974,A -85,B 0,C 180,E1 -5530.382,E2 -5530.382} C_VEL
LIN {X 0,Y 509.825,Z 129.975,A -85,B 0,C 180,E1 -5533.062,E2 -5533.062} C_VEL
LIN {X 0,Y 509.824,Z 129.982,A -85,B 0,C 180,E1 -5535.793,E2 -5535.793} C_VEL
LIN {X 0,Y 509.856,Z 129.97,A -85,B 0,C 180,E1 -5538.574,E2 -5538.574} C_VEL
LIN {X 0,Y 509.851,Z 129.976,A -85,B 0,C 180,E1 -5541.786,E2 -5541.786} C_VEL
LIN {X 0,Y 509.83,Z 129.974,A -85,B 0,C 180,E1 -5544.622,E2 -5544.622} C_VEL
LIN {X 0,Y 509.86,Z 129.978,A -85,B 0,C 180,E1 -5547.481,E2 -5547.481} C_VEL
LIN {X 0,Y 509.858,Z 129.97,A -85,B 0,C 180,E1 -5550.274,E2 -5550.274} C_VEL
LIN {X 0,Y 509.884,Z 129.97,A -85,B 0,C 180,E1 -5552.944,E2 -5552.944} C_VEL
LIN {X 0,Y 509.865,Z 129.973,A -85,B 0,C 180,E1 -5555.574,E2 -5555.574} C_VEL
LIN {X 0,Y 509.85,Z 129.977,A -85,B 0,C 180,E1 -5558.998,E2 -5558.998} C_VEL
LIN {X 0,Y 509.861,Z 129.973,A -85,B 0,C 180,E1 -5561.516,E2 -5561.516} C_VEL
LIN {X 0,Y 509.911,Z 129.969,A -85,B 0,C 180,E1 -5564.819,E2 -5564.819} C_VEL
LIN {X 0,Y 509.901,Z 129.965,A -85,B 0,C 180,E1 -5568.124,E2 -5568.124} C_VEL
LIN {X 0,Y 509.904,Z 129.967,A -85,B 0,C 180,E1 -5571.279,E2 -5571.279} C_VEL
LIN {X 0,Y 509.977,Z 129.959,A -85,B 0,C 180,E1 -5574.464,E2 -5574.464} C_VEL
LIN {X 0,Y 510.055,Z 129.945,A -85,B 0,C 180,E1 -5577.631,E2 -5577.631} C_VEL
LIN {X 0,Y 510.064,Z 129.951,A -85,B 0,C 180,E1 -5580.789,E2 -5580.789} C_VEL
LIN {X 0,Y 509.952,Z 129.96,A -85,B 0,C 180,E1 -5583.16,E2 -5583.16} C_VEL
LIN {X 0,Y 509.954,Z 129.964,A -85,B 0,C 180,E1 -5586.33,E2 -5586.33} C_VEL
LIN {X 0,Y 509.911,Z 129.969,A -85,B 0,C 180,E1 -5588.72,E2 -5588.72} C_VEL
LIN {X 0,Y 509.904,Z 129.967,A -85,B 0,C 180,E1 -5591.931,E2 -5591.931} C_VEL
LIN {X 0,Y 509.894,Z 129.965,A -85,B 0,C 180,E1 -5595.242,E2 -5595.242} C_VEL
LIN {X 0,Y 509.86,Z 129.975,A -85,B 0,C 180,E1 -5598.484,E2 -5598.484} C_VEL
LIN {X 0,Y 509.849,Z 129.971,A -85,B 0,C 180,E1 -5601.002,E2 -5601.002} C_VEL
LIN {X 0,Y 509.822,Z 129.976,A -85,B 0,C 180,E1 -5603.564,E2 -5603.564} C_VEL
LIN {X 0,Y 509.909,Z 129.968,A -85,B 0,C 180,E1 -5606.378,E2 -5606.378} C_VEL
LIN {X 0,Y 509.871,Z 129.969,A -85,B 0,C 180,E1 -5608.844,E2 -5608.844} C_VEL
LIN {X 0,Y 509.819,Z 129.978,A -85,B 0,C 180,E1 -5611.59,E2 -5611.59} C_VEL
LIN {X 0,Y 509.846,Z 129.974,A -85,B 0,C 180,E1 -5614.414,E2 -5614.414} C_VEL
LIN {X 0,Y 509.816,Z 129.977,A -85,B 0,C 180,E1 -5617.341,E2 -5617.341} C_VEL
LIN {X 0,Y 509.837,Z 129.974,A -85,B 0,C 180,E1 -5620.382,E2 -5620.382} C_VEL
LIN {X 0,Y 509.823,Z 129.975,A -85,B 0,C 180,E1 -5623.062,E2 -5623.062} C_VEL
LIN {X 0,Y 509.822,Z 129.981,A -85,B 0,C 180,E1 -5625.793,E2 -5625.793} C_VEL
LIN {X 0,Y 509.854,Z 129.97,A -85,B 0,C 180,E1 -5628.575,E2 -5628.575} C_VEL
LIN {X 0,Y 509.85,Z 129.976,A -85,B 0,C 180,E1 -5631.787,E2 -5631.787} C_VEL
LIN {X 0,Y 509.819,Z 129.98,A -85,B 0,C 180,E1 -5633.736,E2 -5633.736} C_VEL
LIN {X 0,Y 509.151,Z 130.06,A -85,B 0,C 180,E1 -5634.396,E2 -5634.396} C_VEL
LIN {X 0,Y 506.338,Z 130.417,A -85,B 0,C 180,E1 -5635.468,E2 -5635.468} C_VEL
LIN {X 0,Y 503.95,Z 130.713,A -85,B 0,C 180,E1 -5636.331,E2 -5636.331} C_VEL
LIN {X 0,Y 502.903,Z 130.84,A -85,B 0,C 180,E1 -5636.998,E2 -5636.998} C_VEL
LIN {X 0,Y 502.805,Z 130.85,A -85,B 0,C 180,E1 -5637.223,E2 -5637.223} C_VEL
LIN {X 0,Y 502.813,Z 130.848,A -85,B 0,C 180,E1 -5640.065,E2 -5640.065} C_VEL
LIN {X 0,Y 502.83,Z 130.846,A -85,B 0,C 180,E1 -5642.533,E2 -5642.533} C_VEL
LIN {X 0,Y 502.826,Z 130.853,A -85,B 0,C 180,E1 -5645.299,E2 -5645.299} C_VEL
LIN {X 0,Y 502.779,Z 130.853,A -85,B 0,C 180,E1 -5647.827,E2 -5647.827} C_VEL
LIN {X 0,Y 502.823,Z 130.847,A -85,B 0,C 180,E1 -5650.4,E2 -5650.4} C_VEL
LIN {X 0,Y 502.819,Z 130.854,A -85,B 0,C 180,E1 -5652.931,E2 -5652.931} C_VEL
LIN {X 0,Y 502.843,Z 130.846,A -85,B 0,C 180,E1 -5655.429,E2 -5655.429} C_VEL
LIN {X 0,Y 502.877,Z 130.846,A -85,B 0,C 180,E1 -5658.717,E2 -5658.717} C_VEL
LIN {X 0,Y 502.881,Z 130.839,A -85,B 0,C 180,E1 -5661.966,E2 -5661.966} C_VEL
LIN {X 0,Y 502.93,Z 130.836,A -85,B 0,C 180,E1 -5664.387,E2 -5664.387} C_VEL
LIN {X 0,Y 503.025,Z 130.824,A -85,B 0,C 180,E1 -5667.598,E2 -5667.598} C_VEL
LIN {X 0,Y 503.031,Z 130.918,A -85,B 0,C 180,E1 -5670.651,E2 -5670.651} C_VEL
LIN {X 0,Y 503.536,Z 137.552,A -85,B 0,C 180,E1 -5672,E2 -5672} C_VEL
LIN {X 0,Y 503.258,Z 148.944,A -85,B 0,C 180,E1 -5674.255,E2 -5674.255} C_VEL
LIN {X 0,Y 505.362,Z 159.457,A -85,B 0,C 180,E1 -5674.487,E2 -5674.487} C_VEL
LIN {X 0,Y 504.845,Z 255.914,A -85,B 0,C 180,E1 -5675.893,E2 -5675.893} C_VEL
LIN {X 0,Y 504.641,Z 269.043,A -85,B 0,C 180,E1 -5676.246,E2 -5676.246} C_VEL
LIN {X 0,Y 504.415,Z 281.65,A -85,B 0,C 180,E1 -5676.751,E2 -5676.751} C_VEL
LIN {X 0,Y 504.115,Z 294.204,A -85,B 0,C 180,E1 -5677.443,E2 -5677.443} C_VEL
LIN {X 0,Y 503.779,Z 305.17,A -85,B 0,C 180,E1 -5678.221,E2 -5678.221} C_VEL
LIN {X 0,Y 503.415,Z 315.546,A -85,B 0,C 180,E1 -5679.138,E2 -5679.138} C_VEL
LIN {X 0,Y 503.101,Z 324.032,A -85,B 0,C 180,E1 -5680.057,E2 -5680.057} C_VEL
LIN {X 0,Y 502.821,Z 333.207,A -85,B 0,C 180,E1 -5681.285,E2 -5681.285} C_VEL
LIN {X 0,Y 502.557,Z 340.623,A -85,B 0,C 180,E1 -5682.519,E2 -5682.519} C_VEL
LIN {X 0,Y 502.38,Z 346.56,A -85,B 0,C 180,E1 -5683.758,E2 -5683.758} C_VEL
LIN {X 0,Y 502.269,Z 351.512,A -85,B 0,C 180,E1 -5685.098,E2 -5685.098} C_VEL
LIN {X 0,Y 502.143,Z 354.752,A -85,B 0,C 180,E1 -5686.256,E2 -5686.256} C_VEL
LIN {X 0,Y 502.058,Z 357.694,A -85,B 0,C 180,E1 -5687.845,E2 -5687.845} C_VEL
LIN {X 0,Y 502.063,Z 358.714,A -85,B 0,C 180,E1 -5688.782,E2 -5688.782} C_VEL
LIN {X 0,Y 502.062,Z 359.164,A -85,B 0,C 180,E1 -5690.301,E2 -5690.301} C_VEL
LIN {X 0,Y 502.042,Z 358.699,A -85,B 0,C 180,E1 -5691.344,E2 -5691.344} C_VEL
LIN {X 0,Y 502.076,Z 357.356,A -85,B 0,C 180,E1 -5692.503,E2 -5692.503} C_VEL
LIN {X 0,Y 502.212,Z 354.52,A -85,B 0,C 180,E1 -5693.943,E2 -5693.943} C_VEL
LIN {X 0,Y 502.276,Z 350.674,A -85,B 0,C 180,E1 -5695.263,E2 -5695.263} C_VEL
LIN {X 0,Y 502.426,Z 345.481,A -85,B 0,C 180,E1 -5696.591,E2 -5696.591} C_VEL
LIN {X 0,Y 502.639,Z 338.742,A -85,B 0,C 180,E1 -5697.931,E2 -5697.931} C_VEL
LIN {X 0,Y 502.867,Z 331.66,A -85,B 0,C 180,E1 -5699.056,E2 -5699.056} C_VEL
LIN {X 0,Y 503.18,Z 322.856,A -85,B 0,C 180,E1 -5700.187,E2 -5700.187} C_VEL
LIN {X 0,Y 503.529,Z 312.374,A -85,B 0,C 180,E1 -5701.274,E2 -5701.274} C_VEL
LIN {X 0,Y 503.898,Z 302.167,A -85,B 0,C 180,E1 -5702.123,E2 -5702.123} C_VEL
LIN {X 0,Y 504.225,Z 291.901,A -85,B 0,C 180,E1 -5702.81,E2 -5702.81} C_VEL
LIN {X 0,Y 504.52,Z 279.798,A -85,B 0,C 180,E1 -5703.441,E2 -5703.441} C_VEL
LIN {X 0,Y 504.779,Z 267.766,A -85,B 0,C 180,E1 -5703.903,E2 -5703.903} C_VEL
LIN {X 0,Y 504.907,Z 254.665,A -85,B 0,C 180,E1 -5704.239,E2 -5704.239} C_VEL
LIN {X 0,Y 505.368,Z 159.355,A -85,B 0,C 180,E1 -5705.625,E2 -5705.625} C_VEL
LIN {X 0,Y 503.369,Z 149.014,A -85,B 0,C 180,E1 -5705.862,E2 -5705.862} C_VEL
LIN {X 0,Y 503.557,Z 136.94,A -85,B 0,C 180,E1 -5708.232,E2 -5708.232} C_VEL
LIN {X 0,Y 502.971,Z 131.581,A -85,B 0,C 180,E1 -5709.317,E2 -5709.317} C_VEL
LIN {X 0,Y 502.804,Z 130.857,A -85,B 0,C 180,E1 -5709.493,E2 -5709.493} C_VEL
LIN {X 0,Y 502.771,Z 130.856,A -85,B 0,C 180,E1 -5712.195,E2 -5712.195} C_VEL
LIN {X 0,Y 502.786,Z 130.861,A -85,B 0,C 180,E1 -5715.47,E2 -5715.47} C_VEL
LIN {X 0,Y 502.764,Z 130.863,A -85,B 0,C 180,E1 -5718.929,E2 -5718.929} C_VEL
LIN {X 0,Y 502.789,Z 130.853,A -85,B 0,C 180,E1 -5722.046,E2 -5722.046} C_VEL
LIN {X 0,Y 502.791,Z 130.859,A -85,B 0,C 180,E1 -5725.034,E2 -5725.034} C_VEL
LIN {X 0,Y 502.772,Z 130.855,A -85,B 0,C 180,E1 -5727.915,E2 -5727.915} C_VEL
LIN {X 0,Y 502.789,Z 130.86,A -85,B 0,C 180,E1 -5730.71,E2 -5730.71} C_VEL
LIN {X 0,Y 502.772,Z 130.855,A -85,B 0,C 180,E1 -5733.461,E2 -5733.461} C_VEL
LIN {X 0,Y 502.752,Z 130.859,A -85,B 0,C 180,E1 -5736.084,E2 -5736.084} C_VEL
LIN {X 0,Y 502.755,Z 130.863,A -85,B 0,C 180,E1 -5738.688,E2 -5738.688} C_VEL
LIN {X 0,Y 502.787,Z 130.851,A -85,B 0,C 180,E1 -5741.899,E2 -5741.899} C_VEL
LIN {X 0,Y 502.792,Z 130.852,A -85,B 0,C 180,E1 -5744.683,E2 -5744.683} C_VEL
LIN {X 0,Y 502.84,Z 130.851,A -85,B 0,C 180,E1 -5748.06,E2 -5748.06} C_VEL
LIN {X 0,Y 502.835,Z 130.845,A -85,B 0,C 180,E1 -5751.156,E2 -5751.156} C_VEL
LIN {X 0,Y 502.866,Z 130.841,A -85,B 0,C 180,E1 -5753.581,E2 -5753.581} C_VEL
LIN {X 0,Y 502.827,Z 130.845,A -85,B 0,C 180,E1 -5756.795,E2 -5756.795} C_VEL
LIN {X 0,Y 502.892,Z 130.838,A -85,B 0,C 180,E1 -5758.399,E2 -5758.399} C_VEL
LIN {X 0,Y 503.003,Z 130.831,A -85,B 0,C 180,E1 -5760,E2 -5760} C_VEL
LIN {X 0,Y 503.009,Z 130.821,A -85,B 0,C 180,E1 -5762.402,E2 -5762.402} C_VEL
LIN {X 0,Y 502.893,Z 130.845,A -85,B 0,C 180,E1 -5765.614,E2 -5765.614} C_VEL
LIN {X 0,Y 502.851,Z 130.844,A -85,B 0,C 180,E1 -5768.034,E2 -5768.034} C_VEL
LIN {X 0,Y 502.878,Z 130.845,A -85,B 0,C 180,E1 -5771.283,E2 -5771.283} C_VEL
LIN {X 0,Y 502.827,Z 130.846,A -85,B 0,C 180,E1 -5774.572,E2 -5774.572} C_VEL
LIN {X 0,Y 502.803,Z 130.848,A -85,B 0,C 180,E1 -5777.909,E2 -5777.909} C_VEL
LIN {X 0,Y 502.832,Z 130.846,A -85,B 0,C 180,E1 -5780.536,E2 -5780.536} C_VEL
LIN {X 0,Y 502.788,Z 130.854,A -85,B 0,C 180,E1 -5783.041,E2 -5783.041} C_VEL
LIN {X 0,Y 502.846,Z 130.844,A -85,B 0,C 180,E1 -5786.556,E2 -5786.556} C_VEL
LIN {X 0,Y 502.812,Z 130.847,A -85,B 0,C 180,E1 -5789.934,E2 -5789.934} C_VEL
LIN {X 0,Y 502.831,Z 130.85,A -85,B 0,C 180,E1 -5793.032,E2 -5793.032} C_VEL
LIN {X 0,Y 502.775,Z 130.854,A -85,B 0,C 180,E1 -5795.951,E2 -5795.951} C_VEL
LIN {X 0,Y 502.796,Z 130.855,A -85,B 0,C 180,E1 -5798.977,E2 -5798.977} C_VEL
LIN {X 0,Y 502.806,Z 130.854,A -85,B 0,C 180,E1 -5802.199,E2 -5802.199} C_VEL
LIN {X 0,Y 502.788,Z 130.852,A -85,B 0,C 180,E1 -5805.47,E2 -5805.47} C_VEL
LIN {X 0,Y 502.797,Z 130.854,A -85,B 0,C 180,E1 -5807.861,E2 -5807.861} C_VEL
LIN {X 0,Y 502.804,Z 130.851,A -85,B 0,C 180,E1 -5811.024,E2 -5811.024} C_VEL
LIN {X 0,Y 502.774,Z 130.861,A -85,B 0,C 180,E1 -5814.17,E2 -5814.17} C_VEL
LIN {X 0,Y 502.835,Z 130.848,A -85,B 0,C 180,E1 -5816.993,E2 -5816.993} C_VEL
LIN {X 0,Y 502.817,Z 130.855,A -85,B 0,C 180,E1 -5820.065,E2 -5820.065} C_VEL
LIN {X 0,Y 502.83,Z 130.851,A -85,B 0,C 180,E1 -5822.533,E2 -5822.533} C_VEL
LIN {X 0,Y 502.866,Z 130.862,A -85,B 0,C 180,E1 -5824.548,E2 -5824.548} C_VEL
LIN {X 0,Y 504.602,Z 140.404,A -85,B 0,C 180,E1 -5826.177,E2 -5826.177} C_VEL
LIN {X 0,Y 504.08,Z 158.772,A -85,B 0,C 180,E1 -5829.089,E2 -5829.089} C_VEL
LIN {X 0,Y 503.52,Z 179.607,A -85,B 0,C 180,E1 -5832.327,E2 -5832.327} C_VEL
LIN {X 0,Y 503.194,Z 191.688,A -85,B 0,C 180,E1 -5834.178,E2 -5834.178} C_VEL
LIN {X 0,Y 505.327,Z 207.477,A -85,B 0,C 180,E1 -5834.477,E2 -5834.477} C_VEL
LIN {X 0,Y 504.837,Z 300.028,A -85,B 0,C 180,E1 -5835.822,E2 -5835.822} C_VEL
LIN {X 0,Y 504.575,Z 312.627,A -85,B 0,C 180,E1 -5836.149,E2 -5836.149} C_VEL
LIN {X 0,Y 504.214,Z 325.61,A -85,B 0,C 180,E1 -5836.652,E2 -5836.652} C_VEL
LIN {X 0,Y 503.84,Z 337.85,A -85,B 0,C 180,E1 -5837.302,E2 -5837.302} C_VEL
LIN {X 0,Y 503.489,Z 349.595,A -85,B 0,C 180,E1 -5838.118,E2 -5838.118} C_VEL
LIN {X 0,Y 503.138,Z 360.086,A -85,B 0,C 180,E1 -5839.028,E2 -5839.028} C_VEL
LIN {X 0,Y 502.814,Z 368.667,A -85,B 0,C 180,E1 -5839.938,E2 -5839.938} C_VEL
LIN {X 0,Y 502.595,Z 376.592,A -85,B 0,C 180,E1 -5840.949,E2 -5840.949} C_VEL
LIN {X 0,Y 502.364,Z 384.342,A -85,B 0,C 180,E1 -5842.16,E2 -5842.16} C_VEL
LIN {X 0,Y 502.216,Z 391.487,A -85,B 0,C 180,E1 -5843.572,E2 -5843.572} C_VEL
LIN {X 0,Y 502.17,Z 396.245,A -85,B 0,C 180,E1 -5844.78,E2 -5844.78} C_VEL
LIN {X 0,Y 502.14,Z 399.881,A -85,B 0,C 180,E1 -5845.987,E2 -5845.987} C_VEL
LIN {X 0,Y 502.137,Z 401.759,A -85,B 0,C 180,E1 -5846.79,E2 -5846.79} C_VEL
LIN {X 0,Y 502.125,Z 403.166,A -85,B 0,C 180,E1 -5847.593,E2 -5847.593} C_VEL
LIN {X 0,Y 502.001,Z 404.783,A -85,B 0,C 180,E1 -5849.198,E2 -5849.198} C_VEL
LIN {X 0,Y 501.997,Z 405.004,A -85,B 0,C 180,E1 -5850,E2 -5850} C_VEL
LIN {X 0,Y 502.037,Z 404.185,A -85,B 0,C 180,E1 -5851.604,E2 -5851.604} C_VEL
LIN {X 0,Y 502.125,Z 403.192,A -85,B 0,C 180,E1 -5852.406,E2 -5852.406} C_VEL
LIN {X 0,Y 502.137,Z 401.791,A -85,B 0,C 180,E1 -5853.209,E2 -5853.209} C_VEL
LIN {X 0,Y 502.101,Z 398.842,A -85,B 0,C 180,E1 -5854.415,E2 -5854.415} C_VEL
LIN {X 0,Y 502.189,Z 394.853,A -85,B 0,C 180,E1 -5855.622,E2 -5855.622} C_VEL
LIN {X 0,Y 502.281,Z 388.814,A -85,B 0,C 180,E1 -5857.012,E2 -5857.012} C_VEL
LIN {X 0,Y 502.445,Z 382.006,A -85,B 0,C 180,E1 -5858.243,E2 -5858.243} C_VEL
LIN {X 0,Y 502.684,Z 373.687,A -85,B 0,C 180,E1 -5859.455,E2 -5859.455} C_VEL
LIN {X 0,Y 502.949,Z 365.155,A -85,B 0,C 180,E1 -5860.466,E2 -5860.466} C_VEL
LIN {X 0,Y 503.307,Z 354.607,A -85,B 0,C 180,E1 -5861.477,E2 -5861.477} C_VEL
LIN {X 0,Y 503.659,Z 342.959,A -85,B 0,C 180,E1 -5862.372,E2 -5862.372} C_VEL
LIN {X 0,Y 504.081,Z 330.764,A -85,B 0,C 180,E1 -5863.095,E2 -5863.095} C_VEL
LIN {X 0,Y 504.354,Z 318.304,A -85,B 0,C 180,E1 -5863.652,E2 -5863.652} C_VEL
LIN {X 0,Y 504.684,Z 305.442,A -85,B 0,C 180,E1 -5864.053,E2 -5864.053} C_VEL
LIN {X 0,Y 504.876,Z 289.983,A -85,B 0,C 180,E1 -5864.331,E2 -5864.331} C_VEL
LIN {X 0,Y 505.174,Z 205.39,A -85,B 0,C 180,E1 -5865.547,E2 -5865.547} C_VEL
LIN {X 0,Y 503.202,Z 191.79,A -85,B 0,C 180,E1 -5865.819,E2 -5865.819} C_VEL
LIN {X 0,Y 503.751,Z 171.671,A -85,B 0,C 180,E1 -5868.927,E2 -5868.927} C_VEL
LIN {X 0,Y 504.321,Z 151.409,A -85,B 0,C 180,E1 -5872.102,E2 -5872.102} C_VEL
LIN {X 0,Y 504.627,Z 140.549,A -85,B 0,C 180,E1 -5873.821,E2 -5873.821} C_VEL
LIN {X 0,Y 502.857,Z 130.849,A -85,B 0,C 180,E1 -5875.48,E2 -5875.48} C_VEL
LIN {X 0,Y 502.838,Z 130.851,A -85,B 0,C 180,E1 -5878.373,E2 -5878.373} C_VEL
LIN {X 0,Y 502.795,Z 130.854,A -85,B 0,C 180,E1 -5881.498,E2 -5881.498} C_VEL
LIN {X 0,Y 502.806,Z 130.857,A -85,B 0,C 180,E1 -5883.994,E2 -5883.994} C_VEL
LIN {X 0,Y 502.779,Z 130.852,A -85,B 0,C 180,E1 -5887.177,E2 -5887.177} C_VEL
LIN {X 0,Y 502.789,Z 130.856,A -85,B 0,C 180,E1 -5890.015,E2 -5890.015} C_VEL
LIN {X 0,Y 502.804,Z 130.852,A -85,B 0,C 180,E1 -5892.199,E2 -5892.199} C_VEL
LIN {X 0,Y 502.787,Z 130.856,A -85,B 0,C 180,E1 -5895.47,E2 -5895.47} C_VEL
LIN {X 0,Y 502.82,Z 130.847,A -85,B 0,C 180,E1 -5898.934,E2 -5898.934} C_VEL
LIN {X 0,Y 502.794,Z 130.852,A -85,B 0,C 180,E1 -5902.046,E2 -5902.046} C_VEL
LIN {X 0,Y 502.796,Z 130.852,A -85,B 0,C 180,E1 -5905.034,E2 -5905.034} C_VEL
LIN {X 0,Y 502.782,Z 130.854,A -85,B 0,C 180,E1 -5907.915,E2 -5907.915} C_VEL
LIN {X 0,Y 502.824,Z 130.847,A -85,B 0,C 180,E1 -5910.712,E2 -5910.712} C_VEL
LIN {X 0,Y 502.863,Z 130.848,A -85,B 0,C 180,E1 -5913.439,E2 -5913.439} C_VEL
LIN {X 0,Y 502.786,Z 130.851,A -85,B 0,C 180,E1 -5916.086,E2 -5916.086} C_VEL
LIN {X 0,Y 502.784,Z 130.854,A -85,B 0,C 180,E1 -5918.689,E2 -5918.689} C_VEL
LIN {X 0,Y 502.826,Z 130.853,A -85,B 0,C 180,E1 -5921.248,E2 -5921.248} C_VEL
LIN {X 0,Y 502.849,Z 130.846,A -85,B 0,C 180,E1 -5924.6,E2 -5924.6} C_VEL
LIN {X 0,Y 502.877,Z 130.84,A -85,B 0,C 180,E1 -5928.039,E2 -5928.039} C_VEL
LIN {X 0,Y 502.864,Z 130.846,A -85,B 0,C 180,E1 -5931.156,E2 -5931.156} C_VEL
LIN {X 0,Y 502.93,Z 130.836,A -85,B 0,C 180,E1 -5934.386,E2 -5934.386} C_VEL
LIN {X 0,Y 503.025,Z 130.821,A -85,B 0,C 180,E1 -5937.598,E2 -5937.598} C_VEL
LIN {X 0,Y 503.028,Z 130.822,A -85,B 0,C 180,E1 -5940,E2 -5940} C_VEL
LIN {X 0,Y 503.026,Z 130.826,A -85,B 0,C 180,E1 -5942.402,E2 -5942.402} C_VEL
LIN {X 0,Y 502.933,Z 130.833,A -85,B 0,C 180,E1 -5945.613,E2 -5945.613} C_VEL
LIN {X 0,Y 502.901,Z 130.839,A -85,B 0,C 180,E1 -5948.033,E2 -5948.033} C_VEL
LIN {X 0,Y 502.877,Z 130.84,A -85,B 0,C 180,E1 -5951.283,E2 -5951.283} C_VEL
LIN {X 0,Y 502.844,Z 130.849,A -85,B 0,C 180,E1 -5954.571,E2 -5954.571} C_VEL
LIN {X 0,Y 502.822,Z 130.85,A -85,B 0,C 180,E1 -5957.908,E2 -5957.908} C_VEL
LIN {X 0,Y 502.828,Z 130.85,A -85,B 0,C 180,E1 -5960.536,E2 -5960.536} C_VEL
LIN {X 0,Y 502.787,Z 130.851,A -85,B 0,C 180,E1 -5963.041,E2 -5963.041} C_VEL
LIN {X 0,Y 502.82,Z 130.85,A -85,B 0,C 180,E1 -5965.677,E2 -5965.677} C_VEL
LIN {X 0,Y 502.836,Z 130.849,A -85,B 0,C 180,E1 -5968.373,E2 -5968.373} C_VEL
LIN {X 0,Y 502.792,Z 130.853,A -85,B 0,C 180,E1 -5971.499,E2 -5971.499} C_VEL
LIN {X 0,Y 502.803,Z 130.856,A -85,B 0,C 180,E1 -5973.994,E2 -5973.994} C_VEL
LIN {X 0,Y 502.777,Z 130.853,A -85,B 0,C 180,E1 -5977.178,E2 -5977.178} C_VEL
LIN {X 0,Y 502.787,Z 130.856,A -85,B 0,C 180,E1 -5980.015,E2 -5980.015} C_VEL
LIN {X 0,Y 502.802,Z 130.851,A -85,B 0,C 180,E1 -5982.199,E2 -5982.199} C_VEL
LIN {X 0,Y 502.785,Z 130.857,A -85,B 0,C 180,E1 -5985.47,E2 -5985.47} C_VEL
LIN {X 0,Y 502.818,Z 130.848,A -85,B 0,C 180,E1 -5988.934,E2 -5988.934} C_VEL
LIN {X 0,Y 502.792,Z 130.852,A -85,B 0,C 180,E1 -5992.046,E2 -5992.046} C_VEL
LIN {X 0,Y 502.795,Z 130.853,A -85,B 0,C 180,E1 -5995.034,E2 -5995.034} C_VEL
LIN {X 0,Y 502.805,Z 130.85,A -85,B 0,C 180,E1 -5997.223,E2 -5997.223} C_VEL
LIN {X 0,Y 502.104,Z 130.939,A -85,B 0,C 180,E1 -5997.892,E2 -5997.892} C_VEL
LIN {X 0,Y 499.24,Z 131.296,A -85,B 0,C 180,E1 -5998.978,E2 -5998.978} C_VEL
LIN {X 0,Y 496.846,Z 131.593,A -85,B 0,C 180,E1 -5999.853,E2 -5999.853} C_VEL
LIN {X 0,Y 495.83,Z 131.718,A -85,B 0,C 180,E1 -6000.528,E2 -6000.528} C_VEL
LIN {X 0,Y 495.752,Z 131.729,A -85,B 0,C 180,E1 -6000.757,E2 -6000.757} C_VEL
LIN {X 0,Y 495.79,Z 131.723,A -85,B 0,C 180,E1 -6003.932,E2 -6003.932} C_VEL
LIN {X 0,Y 495.759,Z 131.735,A -85,B 0,C 180,E1 -6007.139,E2 -6007.139} C_VEL
LIN {X 0,Y 495.77,Z 131.725,A -85,B 0,C 180,E1 -6010.11,E2 -6010.11} C_VEL
LIN {X 0,Y 495.764,Z 131.729,A -85,B 0,C 180,E1 -6012.681,E2 -6012.681} C_VEL
LIN {X 0,Y 495.789,Z 131.728,A -85,B 0,C 180,E1 -6015.217,E2 -6015.217} C_VEL
LIN {X 0,Y 495.852,Z 131.719,A -85,B 0,C 180,E1 -6018.555,E2 -6018.555} C_VEL
LIN {X 0,Y 495.836,Z 131.717,A -85,B 0,C 180,E1 -6021.852,E2 -6021.852} C_VEL
LIN {X 0,Y 495.885,Z 131.713,A -85,B 0,C 180,E1 -6024.307,E2 -6024.307} C_VEL
LIN {X 0,Y 495.993,Z 131.7,A -85,B 0,C 180,E1 -6027.564,E2 -6027.564} C_VEL
LIN {X 0,Y 495.999,Z 131.727,A -85,B 0,C 180,E1 -6030.508,E2 -6030.508} C_VEL
LIN {X 0,Y 496.547,Z 139.155,A -85,B 0,C 180,E1 -6032.028,E2 -6032.028} C_VEL
LIN {X 0,Y 496.274,Z 149.232,A -85,B 0,C 180,E1 -6034.035,E2 -6034.035} C_VEL
LIN {X 0,Y 498.576,Z 161.064,A -85,B 0,C 180,E1 -6034.295,E2 -6034.295} C_VEL
LIN {X 0,Y 497.987,Z 255.973,A -85,B 0,C 180,E1 -6035.695,E2 -6035.695} C_VEL
LIN {X 0,Y 497.774,Z 269.183,A -85,B 0,C 180,E1 -6036.053,E2 -6036.053} C_VEL
LIN {X 0,Y 497.524,Z 281.291,A -85,B 0,C 180,E1 -6036.54,E2 -6036.54} C_VEL
LIN {X 0,Y 497.191,Z 293.54,A -85,B 0,C 180,E1 -6037.207,E2 -6037.207} C_VEL
LIN {X 0,Y 496.84,Z 305.197,A -85,B 0,C 180,E1 -6038.037,E2 -6038.037} C_VEL
LIN {X 0,Y 496.46,Z 315.542,A -85,B 0,C 180,E1 -6038.959,E2 -6038.959} C_VEL
LIN {X 0,Y 496.068,Z 324.944,A -85,B 0,C 180,E1 -6039.994,E2 -6039.994} C_VEL
LIN {X 0,Y 495.784,Z 334.009,A -85,B 0,C 180,E1 -6041.24,E2 -6041.24} C_VEL
LIN {X 0,Y 495.496,Z 341.346,A -85,B 0,C 180,E1 -6042.492,E2 -6042.492} C_VEL
LIN {X 0,Y 495.347,Z 346.284,A -85,B 0,C 180,E1 -6043.539,E2 -6043.539} C_VEL
LIN {X 0,Y 495.207,Z 351.083,A -85,B 0,C 180,E1 -6044.801,E2 -6044.801} C_VEL
LIN {X 0,Y 495.092,Z 354.739,A -85,B 0,C 180,E1 -6046.07,E2 -6046.07} C_VEL
LIN {X 0,Y 494.996,Z 357.334,A -85,B 0,C 180,E1 -6047.347,E2 -6047.347} C_VEL
LIN {X 0,Y 494.967,Z 358.497,A -85,B 0,C 180,E1 -6048.203,E2 -6048.203} C_VEL
LIN {X 0,Y 494.975,Z 359.21,A -85,B 0,C 180,E1 -6049.061,E2 -6049.061} C_VEL
LIN {X 0,Y 494.964,Z 359.467,A -85,B 0,C 180,E1 -6050.425,E2 -6050.425} C_VEL
LIN {X 0,Y 494.95,Z 358.741,A -85,B 0,C 180,E1 -6051.665,E2 -6051.665} C_VEL
LIN {X 0,Y 495.012,Z 357.524,A -85,B 0,C 180,E1 -6052.655,E2 -6052.655} C_VEL
LIN {X 0,Y 495.118,Z 355.178,A -85,B 0,C 180,E1 -6053.863,E2 -6053.863} C_VEL
LIN {X 0,Y 495.196,Z 351.487,A -85,B 0,C 180,E1 -6055.2,E2 -6055.2} C_VEL
LIN {X 0,Y 495.387,Z 345.984,A -85,B 0,C 180,E1 -6056.649,E2 -6056.649} C_VEL
LIN {X 0,Y 495.558,Z 339.846,A -85,B 0,C 180,E1 -6057.905,E2 -6057.905} C_VEL
LIN {X 0,Y 495.821,Z 332.947,A -85,B 0,C 180,E1 -6059.044,E2 -6059.044} C_VEL
LIN {X 0,Y 496.161,Z 324.131,A -85,B 0,C 180,E1 -6060.226,E2 -6060.226} C_VEL
LIN {X 0,Y 496.556,Z 313.692,A -85,B 0,C 180,E1 -6061.342,E2 -6061.342} C_VEL
LIN {X 0,Y 496.903,Z 303.522,A -85,B 0,C 180,E1 -6062.22,E2 -6062.22} C_VEL
LIN {X 0,Y 497.312,Z 292.77,A -85,B 0,C 180,E1 -6062.962,E2 -6062.962} C_VEL
LIN {X 0,Y 497.628,Z 281.604,A -85,B 0,C 180,E1 -6063.565,E2 -6063.565} C_VEL
LIN {X 0,Y 497.889,Z 268.591,A -85,B 0,C 180,E1 -6064.086,E2 -6064.086} C_VEL
LIN {X 0,Y 498.05,Z 255.355,A -85,B 0,C 180,E1 -6064.436,E2 -6064.436} C_VEL
LIN {X 0,Y 498.575,Z 160.29,A -85,B 0,C 180,E1 -6065.84,E2 -6065.84} C_VEL
LIN {X 0,Y 496.389,Z 149.357,A -85,B 0,C 180,E1 -6066.091,E2 -6066.091} C_VEL
LIN {X 0,Y 496.562,Z 137.127,A -85,B 0,C 180,E1 -6068.517,E2 -6068.517} C_VEL
LIN {X 0,Y 495.764,Z 131.734,A -85,B 0,C 180,E1 -6069.637,E2 -6069.637} C_VEL
LIN {X 0,Y 495.703,Z 131.739,A -85,B 0,C 180,E1 -6072.886,E2 -6072.886} C_VEL
LIN {X 0,Y 495.722,Z 131.737,A -85,B 0,C 180,E1 -6075.998,E2 -6075.998} C_VEL
LIN {X 0,Y 495.727,Z 131.737,A -85,B 0,C 180,E1 -6079.296,E2 -6079.296} C_VEL
LIN {X 0,Y 495.745,Z 131.734,A -85,B 0,C 180,E1 -6081.408,E2 -6081.408} C_VEL
LIN {X 0,Y 495.743,Z 131.729,A -85,B 0,C 180,E1 -6084.462,E2 -6084.462} C_VEL
LIN {X 0,Y 495.748,Z 131.732,A -85,B 0,C 180,E1 -6087.404,E2 -6087.404} C_VEL
LIN {X 0,Y 495.738,Z 131.733,A -85,B 0,C 180,E1 -6090.252,E2 -6090.252} C_VEL
LIN {X 0,Y 495.737,Z 131.732,A -85,B 0,C 180,E1 -6093.271,E2 -6093.271} C_VEL
LIN {X 0,Y 495.73,Z 131.737,A -85,B 0,C 180,E1 -6096.612,E2 -6096.612} C_VEL
LIN {X 0,Y 495.724,Z 131.732,A -85,B 0,C 180,E1 -6099.342,E2 -6099.342} C_VEL
LIN {X 0,Y 495.735,Z 131.729,A -85,B 0,C 180,E1 -6101.827,E2 -6101.827} C_VEL
LIN {X 0,Y 495.743,Z 131.727,A -85,B 0,C 180,E1 -6105.216,E2 -6105.216} C_VEL
LIN {X 0,Y 495.814,Z 131.72,A -85,B 0,C 180,E1 -6108.554,E2 -6108.554} C_VEL
LIN {X 0,Y 495.81,Z 131.725,A -85,B 0,C 180,E1 -6111.851,E2 -6111.851} C_VEL
LIN {X 0,Y 495.849,Z 131.72,A -85,B 0,C 180,E1 -6114.306,E2 -6114.306} C_VEL
LIN {X 0,Y 495.975,Z 131.702,A -85,B 0,C 180,E1 -6117.564,E2 -6117.564} C_VEL
LIN {X 0,Y 495.973,Z 131.707,A -85,B 0,C 180,E1 -6120,E2 -6120} C_VEL
LIN {X 0,Y 495.976,Z 131.696,A -85,B 0,C 180,E1 -6122.437,E2 -6122.437} C_VEL
LIN {X 0,Y 495.852,Z 131.723,A -85,B 0,C 180,E1 -6125.694,E2 -6125.694} C_VEL
LIN {X 0,Y 495.814,Z 131.719,A -85,B 0,C 180,E1 -6128.149,E2 -6128.149} C_VEL
LIN {X 0,Y 495.853,Z 131.722,A -85,B 0,C 180,E1 -6131.445,E2 -6131.445} C_VEL
LIN {X 0,Y 495.778,Z 131.725,A -85,B 0,C 180,E1 -6134.783,E2 -6134.783} C_VEL
LIN {X 0,Y 495.774,Z 131.722,A -85,B 0,C 180,E1 -6138.235,E2 -6138.235} C_VEL
LIN {X 0,Y 495.777,Z 131.727,A -85,B 0,C 180,E1 -6140.756,E2 -6140.756} C_VEL
LIN {X 0,Y 495.741,Z 131.734,A -85,B 0,C 180,E1 -6143.388,E2 -6143.388} C_VEL
LIN {X 0,Y 495.775,Z 131.726,A -85,B 0,C 180,E1 -6146.738,E2 -6146.738} C_VEL
LIN {X 0,Y 495.761,Z 131.725,A -85,B 0,C 180,E1 -6150.146,E2 -6150.146} C_VEL
LIN {X 0,Y 495.791,Z 131.724,A -85,B 0,C 180,E1 -6153.244,E2 -6153.244} C_VEL
LIN {X 0,Y 495.722,Z 131.733,A -85,B 0,C 180,E1 -6156.088,E2 -6156.088} C_VEL
LIN {X 0,Y 495.76,Z 131.734,A -85,B 0,C 180,E1 -6158.767,E2 -6158.767} C_VEL
LIN {X 0,Y 495.747,Z 131.73,A -85,B 0,C 180,E1 -6161.782,E2 -6161.782} C_VEL
LIN {X 0,Y 495.74,Z 131.731,A -85,B 0,C 180,E1 -6165.141,E2 -6165.141} C_VEL
LIN {X 0,Y 495.753,Z 131.735,A -85,B 0,C 180,E1 -6168.218,E2 -6168.218} C_VEL
LIN {X 0,Y 495.753,Z 131.729,A -85,B 0,C 180,E1 -6171.408,E2 -6171.408} C_VEL
LIN {X 0,Y 495.748,Z 131.732,A -85,B 0,C 180,E1 -6174.462,E2 -6174.462} C_VEL
LIN {X 0,Y 495.77,Z 131.729,A -85,B 0,C 180,E1 -6177.406,E2 -6177.406} C_VEL
LIN {X 0,Y 495.768,Z 131.733,A -85,B 0,C 180,E1 -6180.254,E2 -6180.254} C_VEL
LIN {X 0,Y 495.826,Z 131.724,A -85,B 0,C 180,E1 -6183.251,E2 -6183.251} C_VEL
LIN {X 0,Y 495.836,Z 131.805,A -85,B 0,C 180,E1 -6184.358,E2 -6184.358} C_VEL
LIN {X 0,Y 497.65,Z 141.517,A -85,B 0,C 180,E1 -6186.045,E2 -6186.045} C_VEL
LIN {X 0,Y 497.289,Z 155.022,A -85,B 0,C 180,E1 -6188.224,E2 -6188.224} C_VEL
LIN {X 0,Y 496.591,Z 177.947,A -85,B 0,C 180,E1 -6191.859,E2 -6191.859} C_VEL
LIN {X 0,Y 496.177,Z 191.265,A -85,B 0,C 180,E1 -6193.938,E2 -6193.938} C_VEL
LIN {X 0,Y 498.489,Z 207.372,A -85,B 0,C 180,E1 -6194.257,E2 -6194.257} C_VEL
LIN {X 0,Y 497.974,Z 299.88,A -85,B 0,C 180,E1 -6195.623,E2 -6195.623} C_VEL
LIN {X 0,Y 497.639,Z 313.172,A -85,B 0,C 180,E1 -6195.978,E2 -6195.978} C_VEL
LIN {X 0,Y 497.27,Z 326.487,A -85,B 0,C 180,E1 -6196.514,E2 -6196.514} C_VEL
LIN {X 0,Y 496.883,Z 337.877,A -85,B 0,C 180,E1 -6197.141,E2 -6197.141} C_VEL
LIN {X 0,Y 496.483,Z 349.309,A -85,B 0,C 180,E1 -6197.948,E2 -6197.948} C_VEL
LIN {X 0,Y 496.097,Z 359.792,A -85,B 0,C 180,E1 -6198.871,E2 -6198.871} C_VEL
LIN {X 0,Y 495.797,Z 368.37,A -85,B 0,C 180,E1 -6199.794,E2 -6199.794} C_VEL
LIN {X 0,Y 495.528,Z 376.288,A -85,B 0,C 180,E1 -6200.819,E2 -6200.819} C_VEL
LIN {X 0,Y 495.311,Z 384.029,A -85,B 0,C 180,E1 -6202.048,E2 -6202.048} C_VEL
LIN {X 0,Y 495.129,Z 391.166,A -85,B 0,C 180,E1 -6203.48,E2 -6203.48} C_VEL
LIN {X 0,Y 495.1,Z 395.922,A -85,B 0,C 180,E1 -6204.706,E2 -6204.706} C_VEL
LIN {X 0,Y 495.034,Z 399.556,A -85,B 0,C 180,E1 -6205.929,E2 -6205.929} C_VEL
LIN {X 0,Y 495.057,Z 401.434,A -85,B 0,C 180,E1 -6206.745,E2 -6206.745} C_VEL
LIN {X 0,Y 495.029,Z 402.841,A -85,B 0,C 180,E1 -6207.559,E2 -6207.559} C_VEL
LIN {X 0,Y 494.92,Z 404.459,A -85,B 0,C 180,E1 -6209.186,E2 -6209.186} C_VEL
LIN {X 0,Y 494.914,Z 404.681,A -85,B 0,C 180,E1 -6210,E2 -6210} C_VEL
LIN {X 0,Y 494.964,Z 403.863,A -85,B 0,C 180,E1 -6211.627,E2 -6211.627} C_VEL
LIN {X 0,Y 495.029,Z 402.869,A -85,B 0,C 180,E1 -6212.441,E2 -6212.441} C_VEL
LIN {X 0,Y 495.057,Z 401.468,A -85,B 0,C 180,E1 -6213.255,E2 -6213.255} C_VEL
LIN {X 0,Y 495.006,Z 398.516,A -85,B 0,C 180,E1 -6214.479,E2 -6214.479} C_VEL
LIN {X 0,Y 495.101,Z 394.523,A -85,B 0,C 180,E1 -6215.702,E2 -6215.702} C_VEL
LIN {X 0,Y 495.236,Z 388.376,A -85,B 0,C 180,E1 -6217.133,E2 -6217.133} C_VEL
LIN {X 0,Y 495.371,Z 381.657,A -85,B 0,C 180,E1 -6218.361,E2 -6218.361} C_VEL
LIN {X 0,Y 495.644,Z 373.325,A -85,B 0,C 180,E1 -6219.591,E2 -6219.591} C_VEL
LIN {X 0,Y 495.953,Z 364.773,A -85,B 0,C 180,E1 -6220.615,E2 -6220.615} C_VEL
LIN {X 0,Y 496.303,Z 354.207,A -85,B 0,C 180,E1 -6221.642,E2 -6221.642} C_VEL
LIN {X 0,Y 496.679,Z 342.766,A -85,B 0,C 180,E1 -6222.533,E2 -6222.533} C_VEL
LIN {X 0,Y 497.139,Z 330.31,A -85,B 0,C 180,E1 -6223.281,E2 -6223.281} C_VEL
LIN {X 0,Y 497.454,Z 317.812,A -85,B 0,C 180,E1 -6223.845,E2 -6223.845} C_VEL
LIN {X 0,Y 497.807,Z 304.842,A -85,B 0,C 180,E1 -6224.251,E2 -6224.251} C_VEL
LIN {X 0,Y 498,Z 289.194,A -85,B 0,C 180,E1 -6224.533,E2 -6224.533} C_VEL
LIN {X 0,Y 498.35,Z 206.372,A -85,B 0,C 180,E1 -6225.74,E2 -6225.74} C_VEL
LIN {X 0,Y 496.191,Z 191.484,A -85,B 0,C 180,E1 -6226.041,E2 -6226.041} C_VEL
LIN {X 0,Y 496.784,Z 171.325,A -85,B 0,C 180,E1 -6229.203,E2 -6229.203} C_VEL
LIN {X 0,Y 497.387,Z 151.019,A -85,B 0,C 180,E1 -6232.427,E2 -6232.427} C_VEL
LIN {X 0,Y 497.659,Z 141.506,A -85,B 0,C 180,E1 -6233.954,E2 -6233.954} C_VEL
LIN {X 0,Y 495.803,Z 131.728,A -85,B 0,C 180,E1 -6235.672,E2 -6235.672} C_VEL
LIN {X 0,Y 495.787,Z 131.729,A -85,B 0,C 180,E1 -6238.492,E2 -6238.492} C_VEL
LIN {X 0,Y 495.757,Z 131.733,A -85,B 0,C 180,E1 -6241.725,E2 -6241.725} C_VEL
LIN {X 0,Y 495.77,Z 131.725,A -85,B 0,C 180,E1 -6244.694,E2 -6244.694} C_VEL
LIN {X 0,Y 495.731,Z 131.734,A -85,B 0,C 180,E1 -6247.561,E2 -6247.561} C_VEL
LIN {X 0,Y 495.767,Z 131.725,A -85,B 0,C 180,E1 -6250.7,E2 -6250.7} C_VEL
LIN {X 0,Y 495.729,Z 131.735,A -85,B 0,C 180,E1 -6254.001,E2 -6254.001} C_VEL
LIN {X 0,Y 495.727,Z 131.732,A -85,B 0,C 180,E1 -6257.117,E2 -6257.117} C_VEL
LIN {X 0,Y 495.759,Z 131.73,A -85,B 0,C 180,E1 -6259.953,E2 -6259.953} C_VEL
LIN {X 0,Y 495.728,Z 131.73,A -85,B 0,C 180,E1 -6262.553,E2 -6262.553} C_VEL
LIN {X 0,Y 495.771,Z 131.733,A -85,B 0,C 180,E1 -6265.456,E2 -6265.456} C_VEL
LIN {X 0,Y 495.755,Z 131.727,A -85,B 0,C 180,E1 -6268.363,E2 -6268.363} C_VEL
LIN {X 0,Y 495.787,Z 131.729,A -85,B 0,C 180,E1 -6271.507,E2 -6271.507} C_VEL
LIN {X 0,Y 495.791,Z 131.723,A -85,B 0,C 180,E1 -6273.932,E2 -6273.932} C_VEL
LIN {X 0,Y 495.76,Z 131.734,A -85,B 0,C 180,E1 -6277.139,E2 -6277.139} C_VEL
LIN {X 0,Y 495.771,Z 131.725,A -85,B 0,C 180,E1 -6280.109,E2 -6280.109} C_VEL
LIN {X 0,Y 495.764,Z 131.729,A -85,B 0,C 180,E1 -6282.68,E2 -6282.68} C_VEL
LIN {X 0,Y 495.79,Z 131.728,A -85,B 0,C 180,E1 -6285.217,E2 -6285.217} C_VEL
LIN {X 0,Y 495.852,Z 131.718,A -85,B 0,C 180,E1 -6288.555,E2 -6288.555} C_VEL
LIN {X 0,Y 495.836,Z 131.717,A -85,B 0,C 180,E1 -6291.851,E2 -6291.851} C_VEL
LIN {X 0,Y 495.885,Z 131.713,A -85,B 0,C 180,E1 -6294.306,E2 -6294.306} C_VEL
LIN {X 0,Y 495.993,Z 131.697,A -85,B 0,C 180,E1 -6297.564,E2 -6297.564} C_VEL
LIN {X 0,Y 495.983,Z 131.705,A -85,B 0,C 180,E1 -6300.812,E2 -6300.812} C_VEL
LIN {X 0,Y 495.994,Z 131.703,A -85,B 0,C 180,E1 -6302.436,E2 -6302.436} C_VEL
LIN {X 0,Y 495.889,Z 131.71,A -85,B 0,C 180,E1 -6305.693,E2 -6305.693} C_VEL
LIN {X 0,Y 495.872,Z 131.716,A -85,B 0,C 180,E1 -6308.148,E2 -6308.148} C_VEL
LIN {X 0,Y 495.851,Z 131.715,A -85,B 0,C 180,E1 -6311.445,E2 -6311.445} C_VEL
LIN {X 0,Y 495.789,Z 131.725,A -85,B 0,C 180,E1 -6314.783,E2 -6314.783} C_VEL
LIN {X 0,Y 495.763,Z 131.726,A -85,B 0,C 180,E1 -6317.319,E2 -6317.319} C_VEL
LIN {X 0,Y 495.77,Z 131.729,A -85,B 0,C 180,E1 -6319.89,E2 -6319.89} C_VEL
LIN {X 0,Y 495.758,Z 131.727,A -85,B 0,C 180,E1 -6322.86,E2 -6322.86} C_VEL
LIN {X 0,Y 495.78,Z 131.732,A -85,B 0,C 180,E1 -6326.068,E2 -6326.068} C_VEL
LIN {X 0,Y 495.768,Z 131.726,A -85,B 0,C 180,E1 -6328.815,E2 -6328.815} C_VEL
LIN {X 0,Y 495.754,Z 131.732,A -85,B 0,C 180,E1 -6331.725,E2 -6331.725} C_VEL
LIN {X 0,Y 495.768,Z 131.726,A -85,B 0,C 180,E1 -6334.694,E2 -6334.694} C_VEL
LIN {X 0,Y 495.728,Z 131.735,A -85,B 0,C 180,E1 -6337.562,E2 -6337.562} C_VEL
LIN {X 0,Y 495.765,Z 131.725,A -85,B 0,C 180,E1 -6340.7,E2 -6340.7} C_VEL
LIN {X 0,Y 495.727,Z 131.734,A -85,B 0,C 180,E1 -6344.002,E2 -6344.002} C_VEL
LIN {X 0,Y 495.725,Z 131.733,A -85,B 0,C 180,E1 -6347.117,E2 -6347.117} C_VEL
LIN {X 0,Y 495.757,Z 131.73,A -85,B 0,C 180,E1 -6349.953,E2 -6349.953} C_VEL
LIN {X 0,Y 495.727,Z 131.73,A -85,B 0,C 180,E1 -6352.553,E2 -6352.553} C_VEL
LIN {X 0,Y 495.77,Z 131.733,A -85,B 0,C 180,E1 -6355.456,E2 -6355.456} C_VEL
LIN {X 0,Y 495.753,Z 131.727,A -85,B 0,C 180,E1 -6358.364,E2 -6358.364} C_VEL
LIN {X 0,Y 495.752,Z 131.729,A -85,B 0,C 180,E1 -6360.757,E2 -6360.757} C_VEL
LIN {X 0,Y 495.095,Z 131.816,A -85,B 0,C 180,E1 -6361.436,E2 -6361.436} C_VEL
LIN {X 0,Y 492.239,Z 132.169,A -85,B 0,C 180,E1 -6362.539,E2 -6362.539} C_VEL
LIN {X 0,Y 489.828,Z 132.471,A -85,B 0,C 180,E1 -6363.427,E2 -6363.427} C_VEL
LIN {X 0,Y 488.809,Z 132.593,A -85,B 0,C 180,E1 -6364.114,E2 -6364.114} C_VEL
LIN {X 0,Y 488.735,Z 132.601,A -85,B 0,C 180,E1 -6364.346,E2 -6364.346} C_VEL
LIN {X 0,Y 488.722,Z 132.612,A -85,B 0,C 180,E1 -6367.153,E2 -6367.153} C_VEL
LIN {X 0,Y 488.724,Z 132.603,A -85,B 0,C 180,E1 -6369.811,E2 -6369.811} C_VEL
LIN {X 0,Y 488.714,Z 132.605,A -85,B 0,C 180,E1 -6372.423,E2 -6372.423} C_VEL
LIN {X 0,Y 488.761,Z 132.606,A -85,B 0,C 180,E1 -6375,E2 -6375} C_VEL
LIN {X 0,Y 488.806,Z 132.594,A -85,B 0,C 180,E1 -6378.388,E2 -6378.388} C_VEL
LIN {X 0,Y 488.785,Z 132.595,A -85,B 0,C 180,E1 -6381.733,E2 -6381.733} C_VEL
LIN {X 0,Y 488.842,Z 132.59,A -85,B 0,C 180,E1 -6384.224,E2 -6384.224} C_VEL
LIN {X 0,Y 488.961,Z 132.576,A -85,B 0,C 180,E1 -6387.529,E2 -6387.529} C_VEL
LIN {X 0,Y 488.99,Z 132.784,A -85,B 0,C 180,E1 -6390.412,E2 -6390.412} C_VEL
LIN {X 0,Y 489.572,Z 139.74,A -85,B 0,C 180,E1 -6391.851,E2 -6391.851} C_VEL
LIN {X 0,Y 489.32,Z 149.481,A -85,B 0,C 180,E1 -6393.809,E2 -6393.809} C_VEL
LIN {X 0,Y 491.791,Z 162.683,A -85,B 0,C 180,E1 -6394.098,E2 -6394.098} C_VEL
LIN {X 0,Y 491.106,Z 256.081,A -85,B 0,C 180,E1 -6395.492,E2 -6395.492} C_VEL
LIN {X 0,Y 490.879,Z 269.364,A -85,B 0,C 180,E1 -6395.855,E2 -6395.855} C_VEL
LIN {X 0,Y 490.624,Z 282.048,A -85,B 0,C 180,E1 -6396.374,E2 -6396.374} C_VEL
LIN {X 0,Y 490.299,Z 293.371,A -85,B 0,C 180,E1 -6396.998,E2 -6396.998} C_VEL
LIN {X 0,Y 489.975,Z 304.531,A -85,B 0,C 180,E1 -6397.794,E2 -6397.794} C_VEL
LIN {X 0,Y 489.507,Z 315.539,A -85,B 0,C 180,E1 -6398.775,E2 -6398.775} C_VEL
LIN {X 0,Y 489.128,Z 324.147,A -85,B 0,C 180,E1 -6399.72,E2 -6399.72} C_VEL
LIN {X 0,Y 488.821,Z 332.067,A -85,B 0,C 180,E1 -6400.772,E2 -6400.772} C_VEL
LIN {X 0,Y 488.515,Z 340.212,A -85,B 0,C 180,E1 -6402.118,E2 -6402.118} C_VEL
LIN {X 0,Y 488.298,Z 346.011,A -85,B 0,C 180,E1 -6403.314,E2 -6403.314} C_VEL
LIN {X 0,Y 488.169,Z 350.928,A -85,B 0,C 180,E1 -6404.593,E2 -6404.593} C_VEL
LIN {X 0,Y 488.03,Z 354.703,A -85,B 0,C 180,E1 -6405.88,E2 -6405.88} C_VEL
LIN {X 0,Y 487.932,Z 356.649,A -85,B 0,C 180,E1 -6406.743,E2 -6406.743} C_VEL
LIN {X 0,Y 487.894,Z 358.699,A -85,B 0,C 180,E1 -6408.064,E2 -6408.064} C_VEL
LIN {X 0,Y 487.869,Z 359.706,A -85,B 0,C 180,E1 -6409.349,E2 -6409.349} C_VEL
LIN {X 0,Y 487.88,Z 359.769,A -85,B 0,C 180,E1 -6410.555,E2 -6410.555} C_VEL
LIN {X 0,Y 487.881,Z 358.778,A -85,B 0,C 180,E1 -6411.996,E2 -6411.996} C_VEL
LIN {X 0,Y 487.936,Z 357.531,A -85,B 0,C 180,E1 -6412.886,E2 -6412.886} C_VEL
LIN {X 0,Y 488.077,Z 354.758,A -85,B 0,C 180,E1 -6414.229,E2 -6414.229} C_VEL
LIN {X 0,Y 488.176,Z 350.767,A -85,B 0,C 180,E1 -6415.588,E2 -6415.588} C_VEL
LIN {X 0,Y 488.341,Z 345.924,A -85,B 0,C 180,E1 -6416.839,E2 -6416.839} C_VEL
LIN {X 0,Y 488.572,Z 339.73,A -85,B 0,C 180,E1 -6418.106,E2 -6418.106} C_VEL
LIN {X 0,Y 488.851,Z 332.731,A -85,B 0,C 180,E1 -6419.262,E2 -6419.262} C_VEL
LIN {X 0,Y 489.206,Z 323.736,A -85,B 0,C 180,E1 -6420.462,E2 -6420.462} C_VEL
LIN {X 0,Y 489.635,Z 313.143,A -85,B 0,C 180,E1 -6421.595,E2 -6421.595} C_VEL
LIN {X 0,Y 490.009,Z 303.521,A -85,B 0,C 180,E1 -6422.425,E2 -6422.425} C_VEL
LIN {X 0,Y 490.489,Z 291.673,A -85,B 0,C 180,E1 -6423.235,E2 -6423.235} C_VEL
LIN {X 0,Y 490.82,Z 279.124,A -85,B 0,C 180,E1 -6423.893,E2 -6423.893} C_VEL
LIN {X 0,Y 491.097,Z 266.301,A -85,B 0,C 180,E1 -6424.375,E2 -6424.375} C_VEL
LIN {X 0,Y 491.243,Z 253.118,A -85,B 0,C 180,E1 -6424.69,E2 -6424.69} C_VEL
LIN {X 0,Y 491.847,Z 161.489,A -85,B 0,C 180,E1 -6426.056,E2 -6426.056} C_VEL
LIN {X 0,Y 489.476,Z 149.681,A -85,B 0,C 180,E1 -6426.336,E2 -6426.336} C_VEL
LIN {X 0,Y 489.625,Z 138.309,A -85,B 0,C 180,E1 -6428.613,E2 -6428.613} C_VEL
LIN {X 0,Y 488.722,Z 132.611,A -85,B 0,C 180,E1 -6429.854,E2 -6429.854} C_VEL
LIN {X 0,Y 488.664,Z 132.616,A -85,B 0,C 180,E1 -6432.821,E2 -6432.821} C_VEL
LIN {X 0,Y 488.688,Z 132.613,A -85,B 0,C 180,E1 -6435.978,E2 -6435.978} C_VEL
LIN {X 0,Y 488.662,Z 132.616,A -85,B 0,C 180,E1 -6438.58,E2 -6438.58} C_VEL
LIN {X 0,Y 488.698,Z 132.611,A -85,B 0,C 180,E1 -6440.949,E2 -6440.949} C_VEL
LIN {X 0,Y 488.669,Z 132.608,A -85,B 0,C 180,E1 -6443.867,E2 -6443.867} C_VEL
LIN {X 0,Y 488.702,Z 132.613,A -85,B 0,C 180,E1 -6446.875,E2 -6446.875} C_VEL
LIN {X 0,Y 488.697,Z 132.609,A -85,B 0,C 180,E1 -6449.779,E2 -6449.779} C_VEL
LIN {X 0,Y 488.696,Z 132.611,A -85,B 0,C 180,E1 -6453.079,E2 -6453.079} C_VEL
LIN {X 0,Y 488.691,Z 132.61,A -85,B 0,C 180,E1 -6455.351,E2 -6455.351} C_VEL
LIN {X 0,Y 488.681,Z 132.608,A -85,B 0,C 180,E1 -6458.043,E2 -6458.043} C_VEL
LIN {X 0,Y 488.684,Z 132.611,A -85,B 0,C 180,E1 -6460.684,E2 -6460.684} C_VEL
LIN {X 0,Y 488.668,Z 132.611,A -85,B 0,C 180,E1 -6463.283,E2 -6463.283} C_VEL
LIN {X 0,Y 488.693,Z 132.607,A -85,B 0,C 180,E1 -6465.849,E2 -6465.849} C_VEL
LIN {X 0,Y 488.775,Z 132.599,A -85,B 0,C 180,E1 -6468.387,E2 -6468.387} C_VEL
LIN {X 0,Y 488.754,Z 132.603,A -85,B 0,C 180,E1 -6471.733,E2 -6471.733} C_VEL
LIN {X 0,Y 488.81,Z 132.597,A -85,B 0,C 180,E1 -6474.224,E2 -6474.224} C_VEL
LIN {X 0,Y 488.941,Z 132.577,A -85,B 0,C 180,E1 -6477.529,E2 -6477.529} C_VEL
LIN {X 0,Y 488.942,Z 132.582,A -85,B 0,C 180,E1 -6480,E2 -6480} C_VEL
LIN {X 0,Y 488.942,Z 132.572,A -85,B 0,C 180,E1 -6482.472,E2 -6482.472} C_VEL
LIN {X 0,Y 488.812,Z 132.598,A -85,B 0,C 180,E1 -6485.776,E2 -6485.776} C_VEL
LIN {X 0,Y 488.761,Z 132.597,A -85,B 0,C 180,E1 -6488.268,E2 -6488.268} C_VEL
LIN {X 0,Y 488.807,Z 132.596,A -85,B 0,C 180,E1 -6491.613,E2 -6491.613} C_VEL
LIN {X 0,Y 488.754,Z 132.602,A -85,B 0,C 180,E1 -6495.001,E2 -6495.001} C_VEL
LIN {X 0,Y 488.746,Z 132.597,A -85,B 0,C 180,E1 -6498.443,E2 -6498.443} C_VEL
LIN {X 0,Y 488.709,Z 132.611,A -85,B 0,C 180,E1 -6501.071,E2 -6501.071} C_VEL
LIN {X 0,Y 488.672,Z 132.611,A -85,B 0,C 180,E1 -6503.747,E2 -6503.747} C_VEL
LIN {X 0,Y 488.725,Z 132.606,A -85,B 0,C 180,E1 -6506.928,E2 -6506.928} C_VEL
LIN {X 0,Y 488.706,Z 132.605,A -85,B 0,C 180,E1 -6510.362,E2 -6510.362} C_VEL
LIN {X 0,Y 488.731,Z 132.602,A -85,B 0,C 180,E1 -6513.483,E2 -6513.483} C_VEL
LIN {X 0,Y 488.684,Z 132.612,A -85,B 0,C 180,E1 -6516.354,E2 -6516.354} C_VEL
LIN {X 0,Y 488.696,Z 132.609,A -85,B 0,C 180,E1 -6519.255,E2 -6519.255} C_VEL
LIN {X 0,Y 488.689,Z 132.615,A -85,B 0,C 180,E1 -6522.526,E2 -6522.526} C_VEL
LIN {X 0,Y 488.704,Z 132.608,A -85,B 0,C 180,E1 -6525.197,E2 -6525.197} C_VEL
LIN {X 0,Y 488.697,Z 132.614,A -85,B 0,C 180,E1 -6528.583,E2 -6528.583} C_VEL
LIN {X 0,Y 488.706,Z 132.608,A -85,B 0,C 180,E1 -6530.947,E2 -6530.947} C_VEL
LIN {X 0,Y 488.672,Z 132.614,A -85,B 0,C 180,E1 -6533.867,E2 -6533.867} C_VEL
LIN {X 0,Y 488.741,Z 132.604,A -85,B 0,C 180,E1 -6536.877,E2 -6536.877} C_VEL
LIN {X 0,Y 488.725,Z 132.609,A -85,B 0,C 180,E1 -6539.781,E2 -6539.781} C_VEL
LIN {X 0,Y 488.794,Z 132.6,A -85,B 0,C 180,E1 -6543.057,E2 -6543.057} C_VEL
LIN {X 0,Y 488.798,Z 132.774,A -85,B 0,C 180,E1 -6544.161,E2 -6544.161} C_VEL
LIN {X 0,Y 490.711,Z 142.626,A -85,B 0,C 180,E1 -6545.909,E2 -6545.909} C_VEL
LIN {X 0,Y 490.395,Z 153.432,A -85,B 0,C 180,E1 -6547.68,E2 -6547.68} C_VEL
LIN {X 0,Y 489.784,Z 169.61,A -85,B 0,C 180,E1 -6550.293,E2 -6550.293} C_VEL
LIN {X 0,Y 489.361,Z 185.761,A -85,B 0,C 180,E1 -6552.878,E2 -6552.878} C_VEL
LIN {X 0,Y 489.217,Z 190.869,A -85,B 0,C 180,E1 -6553.689,E2 -6553.689} C_VEL
LIN {X 0,Y 491.681,Z 208.153,A -85,B 0,C 180,E1 -6554.045,E2 -6554.045} C_VEL
LIN {X 0,Y 491.12,Z 299.726,A -85,B 0,C 180,E1 -6555.418,E2 -6555.418} C_VEL
LIN {X 0,Y 490.774,Z 312.955,A -85,B 0,C 180,E1 -6555.778,E2 -6555.778} C_VEL
LIN {X 0,Y 490.331,Z 326.235,A -85,B 0,C 180,E1 -6556.32,E2 -6556.32} C_VEL
LIN {X 0,Y 489.936,Z 337.718,A -85,B 0,C 180,E1 -6556.963,E2 -6556.963} C_VEL
LIN {X 0,Y 489.477,Z 349.023,A -85,B 0,C 180,E1 -6557.773,E2 -6557.773} C_VEL
LIN {X 0,Y 489.1,Z 359.5,A -85,B 0,C 180,E1 -6558.709,E2 -6558.709} C_VEL
LIN {X 0,Y 488.775,Z 368.072,A -85,B 0,C 180,E1 -6559.646,E2 -6559.646} C_VEL
LIN {X 0,Y 488.466,Z 375.985,A -85,B 0,C 180,E1 -6560.685,E2 -6560.685} C_VEL
LIN {X 0,Y 488.24,Z 383.72,A -85,B 0,C 180,E1 -6561.932,E2 -6561.932} C_VEL
LIN {X 0,Y 488.043,Z 390.855,A -85,B 0,C 180,E1 -6563.385,E2 -6563.385} C_VEL
LIN {X 0,Y 488.009,Z 395.609,A -85,B 0,C 180,E1 -6564.629,E2 -6564.629} C_VEL
LIN {X 0,Y 487.93,Z 399.24,A -85,B 0,C 180,E1 -6565.87,E2 -6565.87} C_VEL
LIN {X 0,Y 487.978,Z 401.117,A -85,B 0,C 180,E1 -6566.697,E2 -6566.697} C_VEL
LIN {X 0,Y 487.937,Z 402.522,A -85,B 0,C 180,E1 -6567.523,E2 -6567.523} C_VEL
LIN {X 0,Y 487.893,Z 403.526,A -85,B 0,C 180,E1 -6568.349,E2 -6568.349} C_VEL
LIN {X 0,Y 487.834,Z 404.358,A -85,B 0,C 180,E1 -6570,E2 -6570} C_VEL
LIN {X 0,Y 487.893,Z 403.535,A -85,B 0,C 180,E1 -6571.651,E2 -6571.651} C_VEL
LIN {X 0,Y 487.937,Z 402.538,A -85,B 0,C 180,E1 -6572.476,E2 -6572.476} C_VEL
LIN {X 0,Y 487.978,Z 401.134,A -85,B 0,C 180,E1 -6573.302,E2 -6573.302} C_VEL
LIN {X 0,Y 487.919,Z 398.177,A -85,B 0,C 180,E1 -6574.544,E2 -6574.544} C_VEL
LIN {X 0,Y 487.995,Z 394.178,A -85,B 0,C 180,E1 -6575.786,E2 -6575.786} C_VEL
LIN {X 0,Y 488.17,Z 388.023,A -85,B 0,C 180,E1 -6577.237,E2 -6577.237} C_VEL
LIN {X 0,Y 488.317,Z 381.296,A -85,B 0,C 180,E1 -6578.483,E2 -6578.483} C_VEL
LIN {X 0,Y 488.578,Z 372.954,A -85,B 0,C 180,E1 -6579.731,E2 -6579.731} C_VEL
LIN {X 0,Y 488.927,Z 364.388,A -85,B 0,C 180,E1 -6580.77,E2 -6580.77} C_VEL
LIN {X 0,Y 489.327,Z 353.809,A -85,B 0,C 180,E1 -6581.81,E2 -6581.81} C_VEL
LIN {X 0,Y 489.733,Z 342.405,A -85,B 0,C 180,E1 -6582.71,E2 -6582.71} C_VEL
LIN {X 0,Y 490.134,Z 331.833,A -85,B 0,C 180,E1 -6583.368,E2 -6583.368} C_VEL
LIN {X 0,Y 490.447,Z 319.923,A -85,B 0,C 180,E1 -6583.941,E2 -6583.941} C_VEL
LIN {X 0,Y 490.871,Z 306.184,A -85,B 0,C 180,E1 -6584.404,E2 -6584.404} C_VEL
LIN {X 0,Y 491.094,Z 293.753,A -85,B 0,C 180,E1 -6584.662,E2 -6584.662} C_VEL
LIN {X 0,Y 491.445,Z 206.692,A -85,B 0,C 180,E1 -6585.951,E2 -6585.951} C_VEL
LIN {X 0,Y 489.192,Z 191.175,A -85,B 0,C 180,E1 -6586.269,E2 -6586.269} C_VEL
LIN {X 0,Y 489.773,Z 172.296,A -85,B 0,C 180,E1 -6589.271,E2 -6589.271} C_VEL
LIN {X 0,Y 490.513,Z 150.614,A -85,B 0,C 180,E1 -6592.759,E2 -6592.759} C_VEL
LIN {X 0,Y 490.654,Z 142.461,A -85,B 0,C 180,E1 -6594.093,E2 -6594.093} C_VEL
LIN {X 0,Y 488.775,Z 132.605,A -85,B 0,C 180,E1 -6595.84,E2 -6595.84} C_VEL
LIN {X 0,Y 488.73,Z 132.606,A -85,B 0,C 180,E1 -6598.695,E2 -6598.695} C_VEL
LIN {X 0,Y 488.694,Z 132.609,A -85,B 0,C 180,E1 -6601.179,E2 -6601.179} C_VEL
LIN {X 0,Y 488.732,Z 132.608,A -85,B 0,C 180,E1 -6604.113,E2 -6604.113} C_VEL
LIN {X 0,Y 488.681,Z 132.609,A -85,B 0,C 180,E1 -6607.159,E2 -6607.159} C_VEL
LIN {X 0,Y 488.719,Z 132.605,A -85,B 0,C 180,E1 -6610.344,E2 -6610.344} C_VEL
LIN {X 0,Y 488.686,Z 132.615,A -85,B 0,C 180,E1 -6613.654,E2 -6613.654} C_VEL
LIN {X 0,Y 488.686,Z 132.608,A -85,B 0,C 180,E1 -6616.345,E2 -6616.345} C_VEL
LIN {X 0,Y 488.734,Z 132.609,A -85,B 0,C 180,E1 -6619.676,E2 -6619.676} C_VEL
LIN {X 0,Y 488.68,Z 132.609,A -85,B 0,C 180,E1 -6622.841,E2 -6622.841} C_VEL
LIN {X 0,Y 488.724,Z 132.606,A -85,B 0,C 180,E1 -6625.886,E2 -6625.886} C_VEL
LIN {X 0,Y 488.691,Z 132.608,A -85,B 0,C 180,E1 -6628.82,E2 -6628.82} C_VEL
LIN {X 0,Y 488.744,Z 132.604,A -85,B 0,C 180,E1 -6631.671,E2 -6631.671} C_VEL
LIN {X 0,Y 488.74,Z 132.601,A -85,B 0,C 180,E1 -6634.444,E2 -6634.444} C_VEL
LIN {X 0,Y 488.723,Z 132.611,A -85,B 0,C 180,E1 -6637.153,E2 -6637.153} C_VEL
LIN {X 0,Y 488.725,Z 132.603,A -85,B 0,C 180,E1 -6639.81,E2 -6639.81} C_VEL
LIN {X 0,Y 488.715,Z 132.605,A -85,B 0,C 180,E1 -6642.423,E2 -6642.423} C_VEL
LIN {X 0,Y 488.762,Z 132.606,A -85,B 0,C 180,E1 -6644.999,E2 -6644.999} C_VEL
LIN {X 0,Y 488.806,Z 132.594,A -85,B 0,C 180,E1 -6648.387,E2 -6648.387} C_VEL
LIN {X 0,Y 488.785,Z 132.595,A -85,B 0,C 180,E1 -6651.733,E2 -6651.733} C_VEL
LIN {X 0,Y 488.842,Z 132.589,A -85,B 0,C 180,E1 -6654.224,E2 -6654.224} C_VEL
LIN {X 0,Y 488.961,Z 132.573,A -85,B 0,C 180,E1 -6657.528,E2 -6657.528} C_VEL
LIN {X 0,Y 488.934,Z 132.583,A -85,B 0,C 180,E1 -6660.823,E2 -6660.823} C_VEL
LIN {X 0,Y 488.961,Z 132.579,A -85,B 0,C 180,E1 -6662.471,E2 -6662.471} C_VEL
LIN {X 0,Y 488.848,Z 132.588,A -85,B 0,C 180,E1 -6665.776,E2 -6665.776} C_VEL
LIN {X 0,Y 488.816,Z 132.596,A -85,B 0,C 180,E1 -6668.266,E2 -6668.266} C_VEL
LIN {X 0,Y 488.805,Z 132.593,A -85,B 0,C 180,E1 -6671.612,E2 -6671.612} C_VEL
LIN {X 0,Y 488.761,Z 132.599,A -85,B 0,C 180,E1 -6675,E2 -6675} C_VEL
LIN {X 0,Y 488.746,Z 132.606,A -85,B 0,C 180,E1 -6678.442,E2 -6678.442} C_VEL
LIN {X 0,Y 488.706,Z 132.605,A -85,B 0,C 180,E1 -6681.071,E2 -6681.071} C_VEL
LIN {X 0,Y 488.679,Z 132.611,A -85,B 0,C 180,E1 -6683.746,E2 -6683.746} C_VEL
LIN {X 0,Y 488.79,Z 132.595,A -85,B 0,C 180,E1 -6686.943,E2 -6686.943} C_VEL
LIN {X 0,Y 488.709,Z 132.608,A -85,B 0,C 180,E1 -6690.363,E2 -6690.363} C_VEL
LIN {X 0,Y 488.734,Z 132.604,A -85,B 0,C 180,E1 -6693.484,E2 -6693.484} C_VEL
LIN {X 0,Y 488.681,Z 132.61,A -85,B 0,C 180,E1 -6696.354,E2 -6696.354} C_VEL
LIN {X 0,Y 488.7,Z 132.607,A -85,B 0,C 180,E1 -6699.254,E2 -6699.254} C_VEL
LIN {X 0,Y 488.706,Z 132.611,A -85,B 0,C 180,E1 -6701.6,E2 -6701.6} C_VEL
LIN {X 0,Y 488.7,Z 132.606,A -85,B 0,C 180,E1 -6704.803,E2 -6704.803} C_VEL
LIN {X 0,Y 488.691,Z 132.613,A -85,B 0,C 180,E1 -6707.475,E2 -6707.475} C_VEL
LIN {X 0,Y 488.732,Z 132.608,A -85,B 0,C 180,E1 -6709.677,E2 -6709.677} C_VEL
LIN {X 0,Y 488.678,Z 132.609,A -85,B 0,C 180,E1 -6712.841,E2 -6712.841} C_VEL
LIN {X 0,Y 488.723,Z 132.605,A -85,B 0,C 180,E1 -6715.887,E2 -6715.887} C_VEL
LIN {X 0,Y 488.69,Z 132.609,A -85,B 0,C 180,E1 -6718.82,E2 -6718.82} C_VEL
LIN {X 0,Y 488.743,Z 132.604,A -85,B 0,C 180,E1 -6721.671,E2 -6721.671} C_VEL
LIN {X 0,Y 488.735,Z 132.601,A -85,B 0,C 180,E1 -6724.346,E2 -6724.346} C_VEL
LIN {X 0,Y 488.087,Z 132.688,A -85,B 0,C 180,E1 -6725.034,E2 -6725.034} C_VEL
LIN {X 0,Y 485.221,Z 133.042,A -85,B 0,C 180,E1 -6726.15,E2 -6726.15} C_VEL
LIN {X 0,Y 482.779,Z 133.35,A -85,B 0,C 180,E1 -6727.05,E2 -6727.05} C_VEL
LIN {X 0,Y 481.723,Z 133.476,A -85,B 0,C 180,E1 -6727.745,E2 -6727.745} C_VEL
LIN {X 0,Y 481.635,Z 133.486,A -85,B 0,C 180,E1 -6727.981,E2 -6727.981} C_VEL
LIN {X 0,Y 481.704,Z 133.478,A -85,B 0,C 180,E1 -6730.393,E2 -6730.393} C_VEL
LIN {X 0,Y 481.678,Z 133.489,A -85,B 0,C 180,E1 -6733.034,E2 -6733.034} C_VEL
LIN {X 0,Y 481.688,Z 133.48,A -85,B 0,C 180,E1 -6735.639,E2 -6735.639} C_VEL
LIN {X 0,Y 481.751,Z 133.472,A -85,B 0,C 180,E1 -6738.215,E2 -6738.215} C_VEL
LIN {X 0,Y 481.74,Z 133.473,A -85,B 0,C 180,E1 -6741.611,E2 -6741.611} C_VEL
LIN {X 0,Y 481.801,Z 133.466,A -85,B 0,C 180,E1 -6744.14,E2 -6744.14} C_VEL
LIN {X 0,Y 481.928,Z 133.453,A -85,B 0,C 180,E1 -6747.493,E2 -6747.493} C_VEL
LIN {X 0,Y 481.96,Z 133.618,A -85,B 0,C 180,E1 -6750.261,E2 -6750.261} C_VEL
LIN {X 0,Y 482.61,Z 140.333,A -85,B 0,C 180,E1 -6751.669,E2 -6751.669} C_VEL
LIN {X 0,Y 482.339,Z 149.728,A -85,B 0,C 180,E1 -6753.577,E2 -6753.577} C_VEL
LIN {X 0,Y 484.92,Z 162.572,A -85,B 0,C 180,E1 -6753.87,E2 -6753.87} C_VEL
LIN {X 0,Y 484.224,Z 257.305,A -85,B 0,C 180,E1 -6755.309,E2 -6755.309} C_VEL
LIN {X 0,Y 483.99,Z 270.284,A -85,B 0,C 180,E1 -6755.677,E2 -6755.677} C_VEL
LIN {X 0,Y 483.711,Z 282.82,A -85,B 0,C 180,E1 -6756.204,E2 -6756.204} C_VEL
LIN {X 0,Y 483.348,Z 294.799,A -85,B 0,C 180,E1 -6756.89,E2 -6756.89} C_VEL
LIN {X 0,Y 482.921,Z 306.695,A -85,B 0,C 180,E1 -6757.772,E2 -6757.772} C_VEL
LIN {X 0,Y 482.512,Z 316.609,A -85,B 0,C 180,E1 -6758.692,E2 -6758.692} C_VEL
LIN {X 0,Y 482.114,Z 325.085,A -85,B 0,C 180,E1 -6759.651,E2 -6759.651} C_VEL
LIN {X 0,Y 481.771,Z 334.242,A -85,B 0,C 180,E1 -6760.932,E2 -6760.932} C_VEL
LIN {X 0,Y 481.441,Z 341.736,A -85,B 0,C 180,E1 -6762.237,E2 -6762.237} C_VEL
LIN {X 0,Y 481.203,Z 347.577,A -85,B 0,C 180,E1 -6763.514,E2 -6763.514} C_VEL
LIN {X 0,Y 481.067,Z 352.22,A -85,B 0,C 180,E1 -6764.813,E2 -6764.813} C_VEL
LIN {X 0,Y 480.916,Z 355.746,A -85,B 0,C 180,E1 -6766.121,E2 -6766.121} C_VEL
LIN {X 0,Y 480.818,Z 357.492,A -85,B 0,C 180,E1 -6766.998,E2 -6766.998} C_VEL
LIN {X 0,Y 480.799,Z 359.152,A -85,B 0,C 180,E1 -6768.172,E2 -6768.172} C_VEL
LIN {X 0,Y 480.767,Z 360.105,A -85,B 0,C 180,E1 -6769.647,E2 -6769.647} C_VEL
LIN {X 0,Y 480.78,Z 360.072,A -85,B 0,C 180,E1 -6770.684,E2 -6770.684} C_VEL
LIN {X 0,Y 480.785,Z 359.659,A -85,B 0,C 180,E1 -6771.435,E2 -6771.435} C_VEL
LIN {X 0,Y 480.857,Z 357.81,A -85,B 0,C 180,E1 -6772.96,E2 -6772.96} C_VEL
LIN {X 0,Y 481.009,Z 354.302,A -85,B 0,C 180,E1 -6774.608,E2 -6774.608} C_VEL
LIN {X 0,Y 481.138,Z 350.03,A -85,B 0,C 180,E1 -6775.99,E2 -6775.99} C_VEL
LIN {X 0,Y 481.368,Z 344.203,A -85,B 0,C 180,E1 -6777.402,E2 -6777.402} C_VEL
LIN {X 0,Y 481.671,Z 336.921,A -85,B 0,C 180,E1 -6778.784,E2 -6778.784} C_VEL
LIN {X 0,Y 482.019,Z 329.198,A -85,B 0,C 180,E1 -6779.959,E2 -6779.959} C_VEL
LIN {X 0,Y 482.439,Z 319.539,A -85,B 0,C 180,E1 -6781.141,E2 -6781.141} C_VEL
LIN {X 0,Y 482.884,Z 308.668,A -85,B 0,C 180,E1 -6782.212,E2 -6782.212} C_VEL
LIN {X 0,Y 483.345,Z 298.044,A -85,B 0,C 180,E1 -6783.043,E2 -6783.043} C_VEL
LIN {X 0,Y 483.816,Z 285.595,A -85,B 0,C 180,E1 -6783.8,E2 -6783.8} C_VEL
LIN {X 0,Y 484.087,Z 273.162,A -85,B 0,C 180,E1 -6784.37,E2 -6784.37} C_VEL
LIN {X 0,Y 484.384,Z 259.9,A -85,B 0,C 180,E1 -6784.778,E2 -6784.778} C_VEL
LIN {X 0,Y 484.515,Z 242.566,A -85,B 0,C 180,E1 -6785.084,E2 -6785.084} C_VEL
LIN {X 0,Y 485.004,Z 162.018,A -85,B 0,C 180,E1 -6786.301,E2 -6786.301} C_VEL
LIN {X 0,Y 482.517,Z 149.992,A -85,B 0,C 180,E1 -6786.596,E2 -6786.596} C_VEL
LIN {X 0,Y 482.673,Z 139.243,A -85,B 0,C 180,E1 -6788.764,E2 -6788.764} C_VEL
LIN {X 0,Y 481.673,Z 133.489,A -85,B 0,C 180,E1 -6790.006,E2 -6790.006} C_VEL
LIN {X 0,Y 481.621,Z 133.496,A -85,B 0,C 180,E1 -6793.302,E2 -6793.302} C_VEL
LIN {X 0,Y 481.652,Z 133.493,A -85,B 0,C 180,E1 -6795.642,E2 -6795.642} C_VEL
LIN {X 0,Y 481.623,Z 133.497,A -85,B 0,C 180,E1 -6798.955,E2 -6798.955} C_VEL
LIN {X 0,Y 481.648,Z 133.487,A -85,B 0,C 180,E1 -6801.994,E2 -6801.994} C_VEL
LIN {X 0,Y 481.681,Z 133.485,A -85,B 0,C 180,E1 -6805.317,E2 -6805.317} C_VEL
LIN {X 0,Y 481.629,Z 133.491,A -85,B 0,C 180,E1 -6808.311,E2 -6808.311} C_VEL
LIN {X 0,Y 481.652,Z 133.488,A -85,B 0,C 180,E1 -6811.216,E2 -6811.216} C_VEL
LIN {X 0,Y 481.626,Z 133.49,A -85,B 0,C 180,E1 -6814.039,E2 -6814.039} C_VEL
LIN {X 0,Y 481.652,Z 133.487,A -85,B 0,C 180,E1 -6816.819,E2 -6816.819} C_VEL
LIN {X 0,Y 481.617,Z 133.489,A -85,B 0,C 180,E1 -6819.499,E2 -6819.499} C_VEL
LIN {X 0,Y 481.645,Z 133.487,A -85,B 0,C 180,E1 -6822.156,E2 -6822.156} C_VEL
LIN {X 0,Y 481.69,Z 133.48,A -85,B 0,C 180,E1 -6824.774,E2 -6824.774} C_VEL
LIN {X 0,Y 481.726,Z 133.479,A -85,B 0,C 180,E1 -6828.215,E2 -6828.215} C_VEL
LIN {X 0,Y 481.712,Z 133.479,A -85,B 0,C 180,E1 -6831.611,E2 -6831.611} C_VEL
LIN {X 0,Y 481.771,Z 133.472,A -85,B 0,C 180,E1 -6834.139,E2 -6834.139} C_VEL
LIN {X 0,Y 481.906,Z 133.453,A -85,B 0,C 180,E1 -6837.493,E2 -6837.493} C_VEL
LIN {X 0,Y 481.911,Z 133.458,A -85,B 0,C 180,E1 -6840,E2 -6840} C_VEL
LIN {X 0,Y 481.907,Z 133.448,A -85,B 0,C 180,E1 -6842.508,E2 -6842.508} C_VEL
LIN {X 0,Y 481.774,Z 133.474,A -85,B 0,C 180,E1 -6845.861,E2 -6845.861} C_VEL
LIN {X 0,Y 481.72,Z 133.473,A -85,B 0,C 180,E1 -6848.389,E2 -6848.389} C_VEL
LIN {X 0,Y 481.753,Z 133.472,A -85,B 0,C 180,E1 -6851.785,E2 -6851.785} C_VEL
LIN {X 0,Y 481.739,Z 133.479,A -85,B 0,C 180,E1 -6855.225,E2 -6855.225} C_VEL
LIN {X 0,Y 481.708,Z 133.475,A -85,B 0,C 180,E1 -6858.722,E2 -6858.722} C_VEL
LIN {X 0,Y 481.647,Z 133.486,A -85,B 0,C 180,E1 -6861.395,E2 -6861.395} C_VEL
LIN {X 0,Y 481.651,Z 133.484,A -85,B 0,C 180,E1 -6864.115,E2 -6864.115} C_VEL
LIN {X 0,Y 481.693,Z 133.483,A -85,B 0,C 180,E1 -6867.126,E2 -6867.126} C_VEL
LIN {X 0,Y 481.668,Z 133.481,A -85,B 0,C 180,E1 -6869.742,E2 -6869.742} C_VEL
LIN {X 0,Y 481.672,Z 133.488,A -85,B 0,C 180,E1 -6872.674,E2 -6872.674} C_VEL
LIN {X 0,Y 481.638,Z 133.487,A -85,B 0,C 180,E1 -6875.71,E2 -6875.71} C_VEL
LIN {X 0,Y 481.668,Z 133.489,A -85,B 0,C 180,E1 -6878.86,E2 -6878.86} C_VEL
LIN {X 0,Y 481.642,Z 133.49,A -85,B 0,C 180,E1 -6882.162,E2 -6882.162} C_VEL
LIN {X 0,Y 481.656,Z 133.485,A -85,B 0,C 180,E1 -6885.542,E2 -6885.542} C_VEL
LIN {X 0,Y 481.651,Z 133.488,A -85,B 0,C 180,E1 -6888.957,E2 -6888.957} C_VEL
LIN {X 0,Y 481.653,Z 133.489,A -85,B 0,C 180,E1 -6891.993,E2 -6891.993} C_VEL
LIN {X 0,Y 481.69,Z 133.479,A -85,B 0,C 180,E1 -6895.318,E2 -6895.318} C_VEL
LIN {X 0,Y 481.647,Z 133.493,A -85,B 0,C 180,E1 -6898.312,E2 -6898.312} C_VEL
LIN {X 0,Y 481.7,Z 133.482,A -85,B 0,C 180,E1 -6901.218,E2 -6901.218} C_VEL
LIN {X 0,Y 481.742,Z 133.609,A -85,B 0,C 180,E1 -6903.929,E2 -6903.929} C_VEL
LIN {X 0,Y 483.754,Z 143.753,A -85,B 0,C 180,E1 -6905.769,E2 -6905.769} C_VEL
LIN {X 0,Y 483.609,Z 151.845,A -85,B 0,C 180,E1 -6907.124,E2 -6907.124} C_VEL
LIN {X 0,Y 482.866,Z 169.373,A -85,B 0,C 180,E1 -6909.999,E2 -6909.999} C_VEL
LIN {X 0,Y 482.374,Z 185.524,A -85,B 0,C 180,E1 -6912.622,E2 -6912.622} C_VEL
LIN {X 0,Y 482.222,Z 190.549,A -85,B 0,C 180,E1 -6913.432,E2 -6913.432} C_VEL
LIN {X 0,Y 484.857,Z 208.516,A -85,B 0,C 180,E1 -6913.812,E2 -6913.812} C_VEL
LIN {X 0,Y 484.255,Z 299.675,A -85,B 0,C 180,E1 -6915.206,E2 -6915.206} C_VEL
LIN {X 0,Y 483.907,Z 312.779,A -85,B 0,C 180,E1 -6915.572,E2 -6915.572} C_VEL
LIN {X 0,Y 483.473,Z 324.868,A -85,B 0,C 180,E1 -6916.068,E2 -6916.068} C_VEL
LIN {X 0,Y 482.99,Z 337.128,A -85,B 0,C 180,E1 -6916.751,E2 -6916.751} C_VEL
LIN {X 0,Y 482.568,Z 347.811,A -85,B 0,C 180,E1 -6917.519,E2 -6917.519} C_VEL
LIN {X 0,Y 482.119,Z 359.209,A -85,B 0,C 180,E1 -6918.544,E2 -6918.544} C_VEL
LIN {X 0,Y 481.737,Z 367.773,A -85,B 0,C 180,E1 -6919.493,E2 -6919.493} C_VEL
LIN {X 0,Y 481.429,Z 375.682,A -85,B 0,C 180,E1 -6920.547,E2 -6920.547} C_VEL
LIN {X 0,Y 481.17,Z 383.412,A -85,B 0,C 180,E1 -6921.813,E2 -6921.813} C_VEL
LIN {X 0,Y 480.964,Z 390.545,A -85,B 0,C 180,E1 -6923.287,E2 -6923.287} C_VEL
LIN {X 0,Y 480.92,Z 395.296,A -85,B 0,C 180,E1 -6924.549,E2 -6924.549} C_VEL
LIN {X 0,Y 480.83,Z 398.924,A -85,B 0,C 180,E1 -6925.809,E2 -6925.809} C_VEL
LIN {X 0,Y 480.9,Z 400.801,A -85,B 0,C 180,E1 -6926.649,E2 -6926.649} C_VEL
LIN {X 0,Y 480.85,Z 402.203,A -85,B 0,C 180,E1 -6927.487,E2 -6927.487} C_VEL
LIN {X 0,Y 480.824,Z 403.206,A -85,B 0,C 180,E1 -6928.325,E2 -6928.325} C_VEL
LIN {X 0,Y 480.757,Z 404.034,A -85,B 0,C 180,E1 -6930,E2 -6930} C_VEL
LIN {X 0,Y 480.824,Z 403.208,A -85,B 0,C 180,E1 -6931.675,E2 -6931.675} C_VEL
LIN {X 0,Y 480.85,Z 402.208,A -85,B 0,C 180,E1 -6932.513,E2 -6932.513} C_VEL
LIN {X 0,Y 480.9,Z 400.801,A -85,B 0,C 180,E1 -6933.351,E2 -6933.351} C_VEL
LIN {X 0,Y 480.837,Z 397.839,A -85,B 0,C 180,E1 -6934.611,E2 -6934.611} C_VEL
LIN {X 0,Y 480.894,Z 393.833,A -85,B 0,C 180,E1 -6935.872,E2 -6935.872} C_VEL
LIN {X 0,Y 481.095,Z 387.669,A -85,B 0,C 180,E1 -6937.344,E2 -6937.344} C_VEL
LIN {X 0,Y 481.268,Z 380.936,A -85,B 0,C 180,E1 -6938.608,E2 -6938.608} C_VEL
LIN {X 0,Y 481.53,Z 372.583,A -85,B 0,C 180,E1 -6939.874,E2 -6939.874} C_VEL
LIN {X 0,Y 481.911,Z 364.003,A -85,B 0,C 180,E1 -6940.929,E2 -6940.929} C_VEL
LIN {X 0,Y 482.333,Z 353.615,A -85,B 0,C 180,E1 -6941.965,E2 -6941.965} C_VEL
LIN {X 0,Y 482.718,Z 343.21,A -85,B 0,C 180,E1 -6942.806,E2 -6942.806} C_VEL
LIN {X 0,Y 483.206,Z 331.388,A -85,B 0,C 180,E1 -6943.564,E2 -6943.564} C_VEL
LIN {X 0,Y 483.627,Z 318.13,A -85,B 0,C 180,E1 -6944.195,E2 -6944.195} C_VEL
LIN {X 0,Y 483.997,Z 304.689,A -85,B 0,C 180,E1 -6944.64,E2 -6944.64} C_VEL
LIN {X 0,Y 484.21,Z 291.177,A -85,B 0,C 180,E1 -6944.902,E2 -6944.902} C_VEL
LIN {X 0,Y 484.617,Z 207.448,A -85,B 0,C 180,E1 -6946.16,E2 -6946.16} C_VEL
LIN {X 0,Y 482.201,Z 190.787,A -85,B 0,C 180,E1 -6946.512,E2 -6946.512} C_VEL
LIN {X 0,Y 482.786,Z 171.882,A -85,B 0,C 180,E1 -6949.561,E2 -6949.561} C_VEL
LIN {X 0,Y 483.559,Z 151.566,A -85,B 0,C 180,E1 -6952.879,E2 -6952.879} C_VEL
LIN {X 0,Y 483.629,Z 143.415,A -85,B 0,C 180,E1 -6954.238,E2 -6954.238} C_VEL
LIN {X 0,Y 481.722,Z 133.483,A -85,B 0,C 180,E1 -6956.014,E2 -6956.014} C_VEL
LIN {X 0,Y 481.677,Z 133.484,A -85,B 0,C 180,E1 -6958.902,E2 -6958.902} C_VEL
LIN {X 0,Y 481.659,Z 133.489,A -85,B 0,C 180,E1 -6962.189,E2 -6962.189} C_VEL
LIN {X 0,Y 481.69,Z 133.48,A -85,B 0,C 180,E1 -6964.682,E2 -6964.682} C_VEL
LIN {X 0,Y 481.656,Z 133.49,A -85,B 0,C 180,E1 -6968.007,E2 -6968.007} C_VEL
LIN {X 0,Y 481.657,Z 133.483,A -85,B 0,C 180,E1 -6971.041,E2 -6971.041} C_VEL
LIN {X 0,Y 481.656,Z 133.484,A -85,B 0,C 180,E1 -6974.458,E2 -6974.458} C_VEL
LIN {X 0,Y 481.648,Z 133.49,A -85,B 0,C 180,E1 -6977.839,E2 -6977.839} C_VEL
LIN {X 0,Y 481.662,Z 133.482,A -85,B 0,C 180,E1 -6980.654,E2 -6980.654} C_VEL
LIN {X 0,Y 481.628,Z 133.493,A -85,B 0,C 180,E1 -6983.376,E2 -6983.376} C_VEL
LIN {X 0,Y 481.677,Z 133.481,A -85,B 0,C 180,E1 -6986.327,E2 -6986.327} C_VEL
LIN {X 0,Y 481.65,Z 133.492,A -85,B 0,C 180,E1 -6989.417,E2 -6989.417} C_VEL
LIN {X 0,Y 481.7,Z 133.478,A -85,B 0,C 180,E1 -6992.168,E2 -6992.168} C_VEL
LIN {X 0,Y 481.713,Z 133.48,A -85,B 0,C 180,E1 -6994.969,E2 -6994.969} C_VEL
LIN {X 0,Y 481.649,Z 133.486,A -85,B 0,C 180,E1 -6997.705,E2 -6997.705} C_VEL
LIN {X 0,Y 481.705,Z 133.478,A -85,B 0,C 180,E1 -7000.393,E2 -7000.393} C_VEL
LIN {X 0,Y 481.679,Z 133.488,A -85,B 0,C 180,E1 -7003.033,E2 -7003.033} C_VEL
LIN {X 0,Y 481.689,Z 133.48,A -85,B 0,C 180,E1 -7005.639,E2 -7005.639} C_VEL
LIN {X 0,Y 481.751,Z 133.472,A -85,B 0,C 180,E1 -7008.215,E2 -7008.215} C_VEL
LIN {X 0,Y 481.74,Z 133.473,A -85,B 0,C 180,E1 -7011.611,E2 -7011.611} C_VEL
LIN {X 0,Y 481.801,Z 133.466,A -85,B 0,C 180,E1 -7014.139,E2 -7014.139} C_VEL
LIN {X 0,Y 481.928,Z 133.45,A -85,B 0,C 180,E1 -7017.492,E2 -7017.492} C_VEL
LIN {X 0,Y 481.886,Z 133.461,A -85,B 0,C 180,E1 -7020.835,E2 -7020.835} C_VEL
LIN {X 0,Y 481.928,Z 133.456,A -85,B 0,C 180,E1 -7022.507,E2 -7022.507} C_VEL
LIN {X 0,Y 481.808,Z 133.465,A -85,B 0,C 180,E1 -7025.86,E2 -7025.86} C_VEL
LIN {X 0,Y 481.761,Z 133.477,A -85,B 0,C 180,E1 -7028.388,E2 -7028.388} C_VEL
LIN {X 0,Y 481.751,Z 133.472,A -85,B 0,C 180,E1 -7031.785,E2 -7031.785} C_VEL
LIN {X 0,Y 481.742,Z 133.472,A -85,B 0,C 180,E1 -7035.224,E2 -7035.224} C_VEL
LIN {X 0,Y 481.708,Z 133.479,A -85,B 0,C 180,E1 -7038.722,E2 -7038.722} C_VEL
LIN {X 0,Y 481.645,Z 133.485,A -85,B 0,C 180,E1 -7041.395,E2 -7041.395} C_VEL
LIN {X 0,Y 481.66,Z 133.491,A -85,B 0,C 180,E1 -7044.114,E2 -7044.114} C_VEL
LIN {X 0,Y 481.745,Z 133.472,A -85,B 0,C 180,E1 -7047.139,E2 -7047.139} C_VEL
LIN {X 0,Y 481.677,Z 133.485,A -85,B 0,C 180,E1 -7049.741,E2 -7049.741} C_VEL
LIN {X 0,Y 481.671,Z 133.482,A -85,B 0,C 180,E1 -7052.674,E2 -7052.674} C_VEL
LIN {X 0,Y 481.635,Z 133.492,A -85,B 0,C 180,E1 -7055.709,E2 -7055.709} C_VEL
LIN {X 0,Y 481.67,Z 133.481,A -85,B 0,C 180,E1 -7058.859,E2 -7058.859} C_VEL
LIN {X 0,Y 481.651,Z 133.49,A -85,B 0,C 180,E1 -7061.913,E2 -7061.913} C_VEL
LIN {X 0,Y 481.654,Z 133.484,A -85,B 0,C 180,E1 -7064.458,E2 -7064.458} C_VEL
LIN {X 0,Y 481.646,Z 133.489,A -85,B 0,C 180,E1 -7067.839,E2 -7067.839} C_VEL
LIN {X 0,Y 481.66,Z 133.483,A -85,B 0,C 180,E1 -7070.654,E2 -7070.654} C_VEL
LIN {X 0,Y 481.626,Z 133.494,A -85,B 0,C 180,E1 -7073.376,E2 -7073.376} C_VEL
LIN {X 0,Y 481.676,Z 133.481,A -85,B 0,C 180,E1 -7076.327,E2 -7076.327} C_VEL
LIN {X 0,Y 481.649,Z 133.491,A -85,B 0,C 180,E1 -7079.418,E2 -7079.418} C_VEL
LIN {X 0,Y 481.699,Z 133.478,A -85,B 0,C 180,E1 -7082.168,E2 -7082.168} C_VEL
LIN {X 0,Y 481.712,Z 133.481,A -85,B 0,C 180,E1 -7084.97,E2 -7084.97} C_VEL
LIN {X 0,Y 481.635,Z 133.486,A -85,B 0,C 180,E1 -7087.981,E2 -7087.981} C_VEL
LIN {X 0,Y 480.968,Z 133.573,A -85,B 0,C 180,E1 -7088.679,E2 -7088.679} C_VEL
LIN {X 0,Y 478.142,Z 133.924,A -85,B 0,C 180,E1 -7089.813,E2 -7089.813} C_VEL
LIN {X 0,Y 475.756,Z 134.223,A -85,B 0,C 180,E1 -7090.728,E2 -7090.728} C_VEL
LIN {X 0,Y 474.73,Z 134.35,A -85,B 0,C 180,E1 -7091.433,E2 -7091.433} C_VEL
LIN {X 0,Y 474.646,Z 134.358,A -85,B 0,C 180,E1 -7091.672,E2 -7091.672} C_VEL
LIN {X 0,Y 474.699,Z 134.352,A -85,B 0,C 180,E1 -7094.544,E2 -7094.544} C_VEL
LIN {X 0,Y 474.704,Z 134.349,A -85,B 0,C 180,E1 -7098.038,E2 -7098.038} C_VEL
LIN {X 0,Y 474.711,Z 134.349,A -85,B 0,C 180,E1 -7101.486,E2 -7101.486} C_VEL
LIN {X 0,Y 474.748,Z 134.351,A -85,B 0,C 180,E1 -7104.904,E2 -7104.904} C_VEL
LIN {X 0,Y 474.894,Z 134.329,A -85,B 0,C 180,E1 -7107.456,E2 -7107.456} C_VEL
LIN {X 0,Y 474.932,Z 134.448,A -85,B 0,C 180,E1 -7110.106,E2 -7110.106} C_VEL
LIN {X 0,Y 475.633,Z 141.967,A -85,B 0,C 180,E1 -7111.694,E2 -7111.694} C_VEL
LIN {X 0,Y 475.389,Z 149.987,A -85,B 0,C 180,E1 -7113.337,E2 -7113.337} C_VEL
LIN {X 0,Y 478.1,Z 163.736,A -85,B 0,C 180,E1 -7113.661,E2 -7113.661} C_VEL
LIN {X 0,Y 477.352,Z 256.961,A -85,B 0,C 180,E1 -7115.095,E2 -7115.095} C_VEL
LIN {X 0,Y 477.101,Z 270.171,A -85,B 0,C 180,E1 -7115.468,E2 -7115.468} C_VEL
LIN {X 0,Y 476.806,Z 283.379,A -85,B 0,C 180,E1 -7116.029,E2 -7116.029} C_VEL
LIN {X 0,Y 476.452,Z 294.516,A -85,B 0,C 180,E1 -7116.671,E2 -7116.671} C_VEL
LIN {X 0,Y 476.048,Z 306.087,A -85,B 0,C 180,E1 -7117.529,E2 -7117.529} C_VEL
LIN {X 0,Y 475.562,Z 316.555,A -85,B 0,C 180,E1 -7118.499,E2 -7118.499} C_VEL
LIN {X 0,Y 475.101,Z 325.956,A -85,B 0,C 180,E1 -7119.58,E2 -7119.58} C_VEL
LIN {X 0,Y 474.717,Z 335.036,A -85,B 0,C 180,E1 -7120.881,E2 -7120.881} C_VEL
LIN {X 0,Y 474.407,Z 341.97,A -85,B 0,C 180,E1 -7122.112,E2 -7122.112} C_VEL
LIN {X 0,Y 474.164,Z 347.307,A -85,B 0,C 180,E1 -7123.282,E2 -7123.282} C_VEL
LIN {X 0,Y 474.016,Z 352.089,A -85,B 0,C 180,E1 -7124.599,E2 -7124.599} C_VEL
LIN {X 0,Y 473.857,Z 355.739,A -85,B 0,C 180,E1 -7125.925,E2 -7125.925} C_VEL
LIN {X 0,Y 473.731,Z 358.327,A -85,B 0,C 180,E1 -7127.26,E2 -7127.26} C_VEL
LIN {X 0,Y 473.708,Z 359.602,A -85,B 0,C 180,E1 -7128.284,E2 -7128.284} C_VEL
LIN {X 0,Y 473.699,Z 360.488,A -85,B 0,C 180,E1 -7129.952,E2 -7129.952} C_VEL
LIN {X 0,Y 473.695,Z 360.327,A -85,B 0,C 180,E1 -7130.86,E2 -7130.86} C_VEL
LIN {X 0,Y 473.692,Z 359.699,A -85,B 0,C 180,E1 -7131.772,E2 -7131.772} C_VEL
LIN {X 0,Y 473.796,Z 357.944,A -85,B 0,C 180,E1 -7133.122,E2 -7133.122} C_VEL
LIN {X 0,Y 473.926,Z 354.996,A -85,B 0,C 180,E1 -7134.533,E2 -7134.533} C_VEL
LIN {X 0,Y 474.074,Z 350.867,A -85,B 0,C 180,E1 -7135.934,E2 -7135.934} C_VEL
LIN {X 0,Y 474.302,Z 345.353,A -85,B 0,C 180,E1 -7137.345,E2 -7137.345} C_VEL
LIN {X 0,Y 474.629,Z 338.152,A -85,B 0,C 180,E1 -7138.767,E2 -7138.767} C_VEL
LIN {X 0,Y 474.974,Z 330.634,A -85,B 0,C 180,E1 -7139.959,E2 -7139.959} C_VEL
LIN {X 0,Y 475.443,Z 321.348,A -85,B 0,C 180,E1 -7141.156,E2 -7141.156} C_VEL
LIN {X 0,Y 475.862,Z 311.09,A -85,B 0,C 180,E1 -7142.215,E2 -7142.215} C_VEL
LIN {X 0,Y 476.385,Z 300.626,A -85,B 0,C 180,E1 -7143.083,E2 -7143.083} C_VEL
LIN {X 0,Y 476.895,Z 288.705,A -85,B 0,C 180,E1 -7143.865,E2 -7143.865} C_VEL
LIN {X 0,Y 477.221,Z 276.086,A -85,B 0,C 180,E1 -7144.486,E2 -7144.486} C_VEL
LIN {X 0,Y 477.539,Z 263.064,A -85,B 0,C 180,E1 -7144.936,E2 -7144.936} C_VEL
LIN {X 0,Y 477.682,Z 250.042,A -85,B 0,C 180,E1 -7145.209,E2 -7145.209} C_VEL
LIN {X 0,Y 478.301,Z 163.298,A -85,B 0,C 180,E1 -7146.537,E2 -7146.537} C_VEL
LIN {X 0,Y 475.613,Z 150.273,A -85,B 0,C 180,E1 -7146.863,E2 -7146.863} C_VEL
LIN {X 0,Y 475.686,Z 140.246,A -85,B 0,C 180,E1 -7148.91,E2 -7148.91} C_VEL
LIN {X 0,Y 474.642,Z 134.364,A -85,B 0,C 180,E1 -7150.21,E2 -7150.21} C_VEL
LIN {X 0,Y 474.587,Z 134.373,A -85,B 0,C 180,E1 -7153.479,E2 -7153.479} C_VEL
LIN {X 0,Y 474.585,Z 134.371,A -85,B 0,C 180,E1 -7156.521,E2 -7156.521} C_VEL
LIN {X 0,Y 474.591,Z 134.369,A -85,B 0,C 180,E1 -7159.34,E2 -7159.34} C_VEL
LIN {X 0,Y 474.606,Z 134.365,A -85,B 0,C 180,E1 -7161.705,E2 -7161.705} C_VEL
LIN {X 0,Y 474.619,Z 134.363,A -85,B 0,C 180,E1 -7164.725,E2 -7164.725} C_VEL
LIN {X 0,Y 474.621,Z 134.362,A -85,B 0,C 180,E1 -7167.787,E2 -7167.787} C_VEL
LIN {X 0,Y 474.592,Z 134.37,A -85,B 0,C 180,E1 -7170.892,E2 -7170.892} C_VEL
LIN {X 0,Y 474.58,Z 134.367,A -85,B 0,C 180,E1 -7173.624,E2 -7173.624} C_VEL
LIN {X 0,Y 474.597,Z 134.368,A -85,B 0,C 180,E1 -7176.653,E2 -7176.653} C_VEL
LIN {X 0,Y 474.586,Z 134.368,A -85,B 0,C 180,E1 -7180.087,E2 -7180.087} C_VEL
LIN {X 0,Y 474.582,Z 134.369,A -85,B 0,C 180,E1 -7182.772,E2 -7182.772} C_VEL
LIN {X 0,Y 474.6,Z 134.36,A -85,B 0,C 180,E1 -7185.42,E2 -7185.42} C_VEL
LIN {X 0,Y 474.685,Z 134.358,A -85,B 0,C 180,E1 -7188.037,E2 -7188.037} C_VEL
LIN {X 0,Y 474.661,Z 134.356,A -85,B 0,C 180,E1 -7191.485,E2 -7191.485} C_VEL
LIN {X 0,Y 474.735,Z 134.348,A -85,B 0,C 180,E1 -7194.052,E2 -7194.052} C_VEL
LIN {X 0,Y 474.871,Z 134.329,A -85,B 0,C 180,E1 -7197.455,E2 -7197.455} C_VEL
LIN {X 0,Y 474.88,Z 134.334,A -85,B 0,C 180,E1 -7200,E2 -7200} C_VEL
LIN {X 0,Y 474.872,Z 134.324,A -85,B 0,C 180,E1 -7202.545,E2 -7202.545} C_VEL
LIN {X 0,Y 474.737,Z 134.349,A -85,B 0,C 180,E1 -7205.948,E2 -7205.948} C_VEL
LIN {X 0,Y 474.669,Z 134.351,A -85,B 0,C 180,E1 -7208.515,E2 -7208.515} C_VEL
LIN {X 0,Y 474.706,Z 134.348,A -85,B 0,C 180,E1 -7211.963,E2 -7211.963} C_VEL
LIN {X 0,Y 474.681,Z 134.355,A -85,B 0,C 180,E1 -7215.767,E2 -7215.767} C_VEL
LIN {X 0,Y 474.662,Z 134.356,A -85,B 0,C 180,E1 -7219.011,E2 -7219.011} C_VEL
LIN {X 0,Y 474.59,Z 134.361,A -85,B 0,C 180,E1 -7221.729,E2 -7221.729} C_VEL
LIN {X 0,Y 474.629,Z 134.36,A -85,B 0,C 180,E1 -7224.495,E2 -7224.495} C_VEL
LIN {X 0,Y 474.639,Z 134.362,A -85,B 0,C 180,E1 -7227.324,E2 -7227.324} C_VEL
LIN {X 0,Y 474.599,Z 134.362,A -85,B 0,C 180,E1 -7230.231,E2 -7230.231} C_VEL
LIN {X 0,Y 474.627,Z 134.361,A -85,B 0,C 180,E1 -7233.222,E2 -7233.222} C_VEL
LIN {X 0,Y 474.591,Z 134.367,A -85,B 0,C 180,E1 -7236.324,E2 -7236.324} C_VEL
LIN {X 0,Y 474.624,Z 134.361,A -85,B 0,C 180,E1 -7239.548,E2 -7239.548} C_VEL
LIN {X 0,Y 474.6,Z 134.368,A -85,B 0,C 180,E1 -7242.233,E2 -7242.233} C_VEL
LIN {X 0,Y 474.618,Z 134.362,A -85,B 0,C 180,E1 -7245.298,E2 -7245.298} C_VEL
LIN {X 0,Y 474.617,Z 134.367,A -85,B 0,C 180,E1 -7248.214,E2 -7248.214} C_VEL
LIN {X 0,Y 474.613,Z 134.363,A -85,B 0,C 180,E1 -7251.543,E2 -7251.543} C_VEL
LIN {X 0,Y 474.625,Z 134.36,A -85,B 0,C 180,E1 -7254.725,E2 -7254.725} C_VEL
LIN {X 0,Y 474.638,Z 134.363,A -85,B 0,C 180,E1 -7257.788,E2 -7257.788} C_VEL
LIN {X 0,Y 474.624,Z 134.363,A -85,B 0,C 180,E1 -7260.885,E2 -7260.885} C_VEL
LIN {X 0,Y 474.694,Z 134.44,A -85,B 0,C 180,E1 -7263.689,E2 -7263.689} C_VEL
LIN {X 0,Y 476.943,Z 146.412,A -85,B 0,C 180,E1 -7265.887,E2 -7265.887} C_VEL
LIN {X 0,Y 476.146,Z 165.094,A -85,B 0,C 180,E1 -7269.027,E2 -7269.027} C_VEL
LIN {X 0,Y 475.534,Z 182.598,A -85,B 0,C 180,E1 -7271.919,E2 -7271.919} C_VEL
LIN {X 0,Y 475.28,Z 190.297,A -85,B 0,C 180,E1 -7273.173,E2 -7273.173} C_VEL
LIN {X 0,Y 478.071,Z 209.295,A -85,B 0,C 180,E1 -7273.576,E2 -7273.576} C_VEL
LIN {X 0,Y 477.421,Z 298.859,A -85,B 0,C 180,E1 -7274.962,E2 -7274.962} C_VEL
LIN {X 0,Y 477.049,Z 312.121,A -85,B 0,C 180,E1 -7275.332,E2 -7275.332} C_VEL
LIN {X 0,Y 476.587,Z 324.856,A -85,B 0,C 180,E1 -7275.863,E2 -7275.863} C_VEL
LIN {X 0,Y 476.059,Z 336.996,A -85,B 0,C 180,E1 -7276.555,E2 -7276.555} C_VEL
LIN {X 0,Y 475.578,Z 348.492,A -85,B 0,C 180,E1 -7277.405,E2 -7277.405} C_VEL
LIN {X 0,Y 475.134,Z 358.968,A -85,B 0,C 180,E1 -7278.373,E2 -7278.373} C_VEL
LIN {X 0,Y 474.726,Z 367.5,A -85,B 0,C 180,E1 -7279.336,E2 -7279.336} C_VEL
LIN {X 0,Y 474.331,Z 376.762,A -85,B 0,C 180,E1 -7280.62,E2 -7280.62} C_VEL
LIN {X 0,Y 474.077,Z 384.232,A -85,B 0,C 180,E1 -7281.904,E2 -7281.904} C_VEL
LIN {X 0,Y 473.896,Z 390.236,A -85,B 0,C 180,E1 -7283.186,E2 -7283.186} C_VEL
LIN {X 0,Y 473.832,Z 394.984,A -85,B 0,C 180,E1 -7284.467,E2 -7284.467} C_VEL
LIN {X 0,Y 473.736,Z 398.609,A -85,B 0,C 180,E1 -7285.746,E2 -7285.746} C_VEL
LIN {X 0,Y 473.806,Z 400.483,A -85,B 0,C 180,E1 -7286.598,E2 -7286.598} C_VEL
LIN {X 0,Y 473.757,Z 402.888,A -85,B 0,C 180,E1 -7288.3,E2 -7288.3} C_VEL
LIN {X 0,Y 473.696,Z 403.498,A -85,B 0,C 180,E1 -7289.15,E2 -7289.15} C_VEL
LIN {X 0,Y 473.683,Z 403.711,A -85,B 0,C 180,E1 -7290,E2 -7290} C_VEL
LIN {X 0,Y 473.757,Z 402.881,A -85,B 0,C 180,E1 -7291.7,E2 -7291.7} C_VEL
LIN {X 0,Y 473.766,Z 401.878,A -85,B 0,C 180,E1 -7292.551,E2 -7292.551} C_VEL
LIN {X 0,Y 473.806,Z 400.466,A -85,B 0,C 180,E1 -7293.401,E2 -7293.401} C_VEL
LIN {X 0,Y 473.76,Z 397.501,A -85,B 0,C 180,E1 -7294.68,E2 -7294.68} C_VEL
LIN {X 0,Y 473.796,Z 393.489,A -85,B 0,C 180,E1 -7295.96,E2 -7295.96} C_VEL
LIN {X 0,Y 473.999,Z 387.315,A -85,B 0,C 180,E1 -7297.454,E2 -7297.454} C_VEL
LIN {X 0,Y 474.18,Z 380.573,A -85,B 0,C 180,E1 -7298.738,E2 -7298.738} C_VEL
LIN {X 0,Y 474.472,Z 372.211,A -85,B 0,C 180,E1 -7300.023,E2 -7300.023} C_VEL
LIN {X 0,Y 474.901,Z 363.618,A -85,B 0,C 180,E1 -7301.092,E2 -7301.092} C_VEL
LIN {X 0,Y 475.333,Z 353.454,A -85,B 0,C 180,E1 -7302.122,E2 -7302.122} C_VEL
LIN {X 0,Y 475.765,Z 342.484,A -85,B 0,C 180,E1 -7303.019,E2 -7303.019} C_VEL
LIN {X 0,Y 476.255,Z 330.885,A -85,B 0,C 180,E1 -7303.766,E2 -7303.766} C_VEL
LIN {X 0,Y 476.685,Z 318.839,A -85,B 0,C 180,E1 -7304.352,E2 -7304.352} C_VEL
LIN {X 0,Y 477.109,Z 305.807,A -85,B 0,C 180,E1 -7304.802,E2 -7304.802} C_VEL
LIN {X 0,Y 477.327,Z 293.544,A -85,B 0,C 180,E1 -7305.068,E2 -7305.068} C_VEL
LIN {X 0,Y 477.811,Z 208.549,A -85,B 0,C 180,E1 -7306.36,E2 -7306.36} C_VEL
LIN {X 0,Y 475.233,Z 190.558,A -85,B 0,C 180,E1 -7306.73,E2 -7306.73} C_VEL
LIN {X 0,Y 475.839,Z 171.469,A -85,B 0,C 180,E1 -7309.859,E2 -7309.859} C_VEL
LIN {X 0,Y 476.619,Z 152.525,A -85,B 0,C 180,E1 -7313.001,E2 -7313.001} C_VEL
LIN {X 0,Y 476.838,Z 145.95,A -85,B 0,C 180,E1 -7314.104,E2 -7314.104} C_VEL
LIN {X 0,Y 474.718,Z 134.355,A -85,B 0,C 180,E1 -7316.203,E2 -7316.203} C_VEL
LIN {X 0,Y 474.621,Z 134.363,A -85,B 0,C 180,E1 -7319.252,E2 -7319.252} C_VEL
LIN {X 0,Y 474.617,Z 134.363,A -85,B 0,C 180,E1 -7322.43,E2 -7322.43} C_VEL
LIN {X 0,Y 474.616,Z 134.363,A -85,B 0,C 180,E1 -7325.469,E2 -7325.469} C_VEL
LIN {X 0,Y 474.613,Z 134.362,A -85,B 0,C 180,E1 -7328.457,E2 -7328.457} C_VEL
LIN {X 0,Y 474.629,Z 134.359,A -85,B 0,C 180,E1 -7330.959,E2 -7330.959} C_VEL
LIN {X 0,Y 474.607,Z 134.365,A -85,B 0,C 180,E1 -7334.105,E2 -7334.105} C_VEL
LIN {X 0,Y 474.615,Z 134.362,A -85,B 0,C 180,E1 -7337.065,E2 -7337.065} C_VEL
LIN {X 0,Y 474.618,Z 134.36,A -85,B 0,C 180,E1 -7340.354,E2 -7340.354} C_VEL
LIN {X 0,Y 474.589,Z 134.37,A -85,B 0,C 180,E1 -7343.676,E2 -7343.676} C_VEL
LIN {X 0,Y 474.625,Z 134.36,A -85,B 0,C 180,E1 -7346.778,E2 -7346.778} C_VEL
LIN {X 0,Y 474.605,Z 134.365,A -85,B 0,C 180,E1 -7349.77,E2 -7349.77} C_VEL
LIN {X 0,Y 474.698,Z 134.351,A -85,B 0,C 180,E1 -7352.68,E2 -7352.68} C_VEL
LIN {X 0,Y 474.656,Z 134.36,A -85,B 0,C 180,E1 -7355.507,E2 -7355.507} C_VEL
LIN {X 0,Y 474.671,Z 134.361,A -85,B 0,C 180,E1 -7359.185,E2 -7359.185} C_VEL
LIN {X 0,Y 474.646,Z 134.357,A -85,B 0,C 180,E1 -7361.884,E2 -7361.884} C_VEL
LIN {X 0,Y 474.7,Z 134.352,A -85,B 0,C 180,E1 -7364.544,E2 -7364.544} C_VEL
LIN {X 0,Y 474.705,Z 134.349,A -85,B 0,C 180,E1 -7368.037,E2 -7368.037} C_VEL
LIN {X 0,Y 474.711,Z 134.35,A -85,B 0,C 180,E1 -7371.486,E2 -7371.486} C_VEL
LIN {X 0,Y 474.748,Z 134.351,A -85,B 0,C 180,E1 -7374.904,E2 -7374.904} C_VEL
LIN {X 0,Y 474.894,Z 134.326,A -85,B 0,C 180,E1 -7377.455,E2 -7377.455} C_VEL
LIN {X 0,Y 474.912,Z 134.324,A -85,B 0,C 180,E1 -7380,E2 -7380} C_VEL
LIN {X 0,Y 474.894,Z 134.333,A -85,B 0,C 180,E1 -7382.544,E2 -7382.544} C_VEL
LIN {X 0,Y 474.771,Z 134.342,A -85,B 0,C 180,E1 -7385.948,E2 -7385.948} C_VEL
LIN {X 0,Y 474.726,Z 134.355,A -85,B 0,C 180,E1 -7388.513,E2 -7388.513} C_VEL
LIN {X 0,Y 474.704,Z 134.352,A -85,B 0,C 180,E1 -7391.962,E2 -7391.962} C_VEL
LIN {X 0,Y 474.699,Z 134.35,A -85,B 0,C 180,E1 -7395.456,E2 -7395.456} C_VEL
LIN {X 0,Y 474.662,Z 134.355,A -85,B 0,C 180,E1 -7399.01,E2 -7399.01} C_VEL
LIN {X 0,Y 474.588,Z 134.366,A -85,B 0,C 180,E1 -7401.729,E2 -7401.729} C_VEL
LIN {X 0,Y 474.64,Z 134.361,A -85,B 0,C 180,E1 -7404.494,E2 -7404.494} C_VEL
LIN {X 0,Y 474.679,Z 134.353,A -85,B 0,C 180,E1 -7407.334,E2 -7407.334} C_VEL
LIN {X 0,Y 474.603,Z 134.362,A -85,B 0,C 180,E1 -7410.81,E2 -7410.81} C_VEL
LIN {X 0,Y 474.637,Z 134.365,A -85,B 0,C 180,E1 -7413.984,E2 -7413.984} C_VEL
LIN {X 0,Y 474.57,Z 134.366,A -85,B 0,C 180,E1 -7416.899,E2 -7416.899} C_VEL
LIN {X 0,Y 474.627,Z 134.365,A -85,B 0,C 180,E1 -7419.648,E2 -7419.648} C_VEL
LIN {X 0,Y 474.613,Z 134.361,A -85,B 0,C 180,E1 -7422.934,E2 -7422.934} C_VEL
LIN {X 0,Y 474.605,Z 134.366,A -85,B 0,C 180,E1 -7425.895,E2 -7425.895} C_VEL
LIN {X 0,Y 474.626,Z 134.361,A -85,B 0,C 180,E1 -7429.041,E2 -7429.041} C_VEL
LIN {X 0,Y 474.609,Z 134.367,A -85,B 0,C 180,E1 -7431.704,E2 -7431.704} C_VEL
LIN {X 0,Y 474.622,Z 134.36,A -85,B 0,C 180,E1 -7434.726,E2 -7434.726} C_VEL
LIN {X 0,Y 474.634,Z 134.361,A -85,B 0,C 180,E1 -7437.788,E2 -7437.788} C_VEL
LIN {X 0,Y 474.622,Z 134.362,A -85,B 0,C 180,E1 -7440.885,E2 -7440.885} C_VEL
LIN {X 0,Y 474.658,Z 134.358,A -85,B 0,C 180,E1 -7443.628,E2 -7443.628} C_VEL
LIN {X 0,Y 474.635,Z 134.36,A -85,B 0,C 180,E1 -7446.642,E2 -7446.642} C_VEL
LIN {X 0,Y 474.654,Z 134.355,A -85,B 0,C 180,E1 -7450.09,E2 -7450.09} C_VEL
LIN {X 0,Y 474.646,Z 134.358,A -85,B 0,C 180,E1 -7451.672,E2 -7451.672} C_VEL
LIN {X 0,Y 473.979,Z 134.441,A -85,B 0,C 180,E1 -7452.381,E2 -7452.381} C_VEL
LIN {X 0,Y 471.132,Z 134.798,A -85,B 0,C 180,E1 -7453.533,E2 -7453.533} C_VEL
LIN {X 0,Y 468.721,Z 135.101,A -85,B 0,C 180,E1 -7454.462,E2 -7454.462} C_VEL
LIN {X 0,Y 467.682,Z 135.229,A -85,B 0,C 180,E1 -7455.179,E2 -7455.179} C_VEL
LIN {X 0,Y 467.596,Z 135.237,A -85,B 0,C 180,E1 -7455.422,E2 -7455.422} C_VEL
LIN {X 0,Y 467.652,Z 135.234,A -85,B 0,C 180,E1 -7458.734,E2 -7458.734} C_VEL
LIN {X 0,Y 467.669,Z 135.227,A -85,B 0,C 180,E1 -7461.357,E2 -7461.357} C_VEL
LIN {X 0,Y 467.724,Z 135.219,A -85,B 0,C 180,E1 -7463.963,E2 -7463.963} C_VEL
LIN {X 0,Y 467.859,Z 135.206,A -85,B 0,C 180,E1 -7467.417,E2 -7467.417} C_VEL
LIN {X 0,Y 467.876,Z 135.269,A -85,B 0,C 180,E1 -7469.946,E2 -7469.946} C_VEL
LIN {X 0,Y 468.663,Z 142.53,A -85,B 0,C 180,E1 -7471.504,E2 -7471.504} C_VEL
LIN {X 0,Y 468.424,Z 150.397,A -85,B 0,C 180,E1 -7473.118,E2 -7473.118} C_VEL
LIN {X 0,Y 471.276,Z 164.798,A -85,B 0,C 180,E1 -7473.447,E2 -7473.447} C_VEL
LIN {X 0,Y 470.454,Z 257.774,A -85,B 0,C 180,E1 -7474.901,E2 -7474.901} C_VEL
